// TIA Portal V20 program export: 1 tag tables, 4 data types, 5 data blocks, 8 code blocks (in call order from the OBs), 4 instance data blocks

VAR_GLOBAL   // PLC tag table "Default tag table"
   Tag_1 AT %I500.0 : Bool;
   Tag_2 AT %I500.1 : Bool;
   Tag_3 AT %I500.2 : Bool;
   Tag_4 AT %I500.3 : Bool;
   Tag_5 AT %I500.6 : Bool;
   Tag_6 AT %I500.7 : Bool;
   Tag_7 AT %I501.0 : Bool;
   Tag_8 AT %I501.1 : Bool;
   Tag_9 AT %I501.2 : Bool;
   Tag_10 AT %I501.3 : Bool;
   Tag_11 AT %I501.4 : Bool;
   Tag_12 AT %I501.5 : Bool;
   Tag_13 AT %I501.6 : Bool;
   Tag_14 AT %I501.7 : Bool;
   Tag_15 AT %I502.1 : Bool;
   Tag_16 AT %I502.2 : Bool;
   Tag_17 AT %I502.3 : Bool;
   Tag_18 AT %I502.4 : Bool;
   Tag_19 AT %I502.5 : Bool;
   Tag_20 AT %I502.6 : Bool;
   Tag_21 AT %I502.7 : Bool;
   Tag_22 AT %I503.0 : Bool;
   Tag_23 AT %I503.1 : Bool;
   Tag_24 AT %I503.2 : Bool;
   Tag_25 AT %I503.3 : Bool;
   Tag_26 AT %I503.4 : Bool;
   Tag_41 AT %IW508 : Word;
   Tag_42 AT %IW528 : Word;
   Tag_43 AT %IW532 : Word;
   Tag_44 AT %IW650 : Word;
   Tag_45 AT %IW64 : Word;
   Tag_46 AT %IW66 : Word;
   Tag_47 AT %IW68 : Word;
   Tag_48 AT %IW70 : Word;
   Tag_49 AT %IW72 : Word;
   Tag_50 AT %IW74 : Word;
   Tag_51 AT %IW76 : Word;
   Tag_52 AT %IW78 : Word;
   Tag_27 AT %Q500.0 : Bool;
   Tag_28 AT %Q500.1 : Bool;
   Tag_29 AT %Q500.2 : Bool;
   Tag_30 AT %Q500.4 : Bool;
   Tag_31 AT %Q500.5 : Bool;
   Tag_32 AT %Q501.0 : Bool;
   Tag_33 AT %Q501.1 : Bool;
   Tag_34 AT %Q501.2 : Bool;
   Tag_35 AT %Q501.3 : Bool;
   Tag_36 AT %Q501.4 : Bool;
   Tag_37 AT %Q501.5 : Bool;
   Tag_38 AT %Q502.0 : Bool;
   Tag_39 AT %Q502.1 : Bool;
   Tag_40 AT %Q502.2 : Bool;
   Tag_53 AT %QW64 : Word;
   Tag_54 AT %QW66 : Word;
   "Clock_0.5Hz" AT %M0.7 : Bool;
   AirStarWord0IN AT %IW80 : Word;
   AirStarWord2IN AT %IW82 : Word;
   AirStarWord0OUT AT %QW68 : Word;
   AirStarWord2OUT AT %QW70 : Word;
   FirstScan AT %M1.0 : Bool;
   AlwaysTrue AT %M1.2 : Bool;
   DI1_SYS_ControlHealthy AT %I0.0 : Bool;   // Safety/control circuit healthy
   DI2_SPR_1 AT %I0.1 : Bool;   // Spare (wired to -X3:1)
   DI3_SYS_CycleStart AT %I0.2 : Bool;   // Cycle start pushbutton (local/remote)
   DI4_SYS_CycleStop AT %I0.3 : Bool;   // Cycle stop pushbutton (NC)
   DI5_SHR_RunFwdFB AT %I0.4 : Bool;   // Shredder running forward feedback
   DI6_SHR_RunRevFB AT %I0.5 : Bool;   // Shredder running reverse feedback
   DI7_SYS_MotorFault AT %I0.6 : Bool;   // Motor fault (soft start fault relay)
   DI8_HPR_LevelHigh AT %I0.7 : Bool;   // Hopper high level sensor
   DI9_IFC_Running AT %I1.0 : Bool;   // Infeed conveyor running feedback
   DI10_DIS_Running AT %I1.1 : Bool;   // Discharge conveyor running feedback
   DI11_PSH_PowerPackRunning AT %I1.2 : Bool;   // Pusher power pack running feedback
   DI12_PSH_HomeLimit AT %I1.3 : Bool;   // Pusher parked/home position
   DI13_PSH_FullTravelLimit AT %I1.4 : Bool;   // Pusher fully extended position
   DI14_PSH_HighPressure AT %I1.5 : Bool;   // Pusher hydraulic high pressure switch
   DI15_SYS_DownstreamRunning AT %I2.0 : Bool;   // Downstream equipment running
   DI16_PSH_LocalRemote AT %I2.1 : Bool;   // Pusher operation local/remote selector
   DI17_SPR_2 AT %I2.2 : Bool;   // Spare (wired to terminal)
   DI18_SPR_3 AT %I2.3 : Bool;   // Spare (wired to terminal)
   DI19_SPR_4 AT %I2.4 : Bool;   // Spare (wired to terminal)
   DI20_SPR_5 AT %I2.5 : Bool;   // Spare (wired to terminal)
   DI21_SPR_6 AT %I2.6 : Bool;   // Spare (wired to terminal)
   DI22_SPR_7 AT %I2.7 : Bool;   // Spare (wired to terminal)
   DQ1_SHR_RunFwd AT %Q0.0 : Bool;   // Run shredder forward command
   DQ2_SHR_RunRev AT %Q0.1 : Bool;   // Run shredder reverse command
   DQ3_PSH_RunPowerPack AT %Q0.2 : Bool;   // Run pusher power pack command
   DQ4_IFC_Run AT %Q0.3 : Bool;   // Run infeed conveyor command
   DQ5_DIS_Run AT %Q0.4 : Bool;   // Run discharge conveyor command
   DQ6_PSH_Extend AT %Q0.5 : Bool;   // Pusher extend solenoid command
   DQ7_PSH_Retract AT %Q0.6 : Bool;   // Pusher retract solenoid command
   DQ8_SYS_InCycle AT %Q0.7 : Bool;   // Machine in-cycle status
   DQ9_SYS_EnableUpstream AT %Q1.0 : Bool;   // Enable upstream equipment (volt-free)
   DQ10_SYS_PreStartSounder AT %Q1.1 : Bool;   // Pre-start warning sounder/beacon
   DQ11_SHR_FaultReset AT %Q2.0 : Bool;   // Soft start motor fault reset
   DQ12_SPR_1 AT %Q2.1 : Bool;   // Spare (relay fitted)
   DQ13_SPR_2 AT %Q2.2 : Bool;   // Spare (relay fitted)
   DQ14_SPR_3 AT %Q2.3 : Bool;   // Spare (relay fitted)
   DQ15_SPR_4 AT %Q2.4 : Bool;   // Spare (relay fitted)
   DQ16_SPR_5 AT %Q2.5 : Bool;   // Spare (relay fitted)
   DQ17_SPR_6 AT %Q2.6 : Bool;   // Spare (wired to -X13:6)
   DQ18_SPR_7 AT %Q2.7 : Bool;   // Spare (wired to -X13:7)
END_VAR

TYPE "MotorFwdRevIOSet"
// stored: IsFailsafeCompliant false
   STRUCT
      InHand : Bool;
      AutoStartSignal : Bool;
      HandStartSignal : Bool;
      RunningFBFwd : Bool;
      RunningFBRev : Bool;
      FaultFB : Bool;
      SystemHealthy : Bool;
      PreStartDone : Bool;
      InhibitMotor : Bool;
      FaultReset : Bool;
      FTTime : Real;
      EnableUPSTime : Real;
      FaultActive : Bool;
      RunFwd : Bool;
      RunRev : Bool;
      UPSEnable : Bool;
      FTR : Bool;
      FTS : Bool;
      HrsRun : UDInt;
      Telemetry : Int;
      Alarm : Word;
      "Name" : String;
      HandIntervention : Bool;
      RecentStart : Bool;
      TryRunMotor : Bool;
      Shutdown : Bool;
      ShutdownComplete : Bool;
      ShutdownTime : Real;
      StopMotor : Bool;
      ReverseDelay : Real;
      ReverseIgnoreFT : Real;
      Reverse : Bool;
      HandReverse : Bool;
   END_STRUCT;
END_TYPE

TYPE "UDT_HopperBlockageIO"
// Caller-visible interface (C-115) for FB_HopperBlockageMonitor. FC_ControlMain writes HopperLevelHigh/PlantRunning/FaultReset in and reads HopperBlockedAlarm/HopperBlockStopReq out (wiring is a separate integration step). Per the Gate-1 supervisory-monitor exemption (NEW-HBA-07) this pure monitor carries no enable/ready/running vocabulary stubs. BlockedTimeThreshold/ClearDebounceTime are this instance's own tunables (C-307), commissioning defaults set as the iDB start values.
// stored: IsFailsafeCompliant false
   STRUCT
      HopperLevelHigh : Bool;   // In (FC_ControlMain, from DB_Input.Hopper_Level_High at integration): hopper high-level sensor - the blockage condition this FB supervises for persistence.
      PlantRunning : Bool;   // In (FC_ControlMain, from DB_Input.Shredder_Run_Fwd_FB OR Shredder_Run_Rev_FB): plant-running gate - the persistence window accrues only while the plant actually runs (Q-HBA-04), so a full hopper at standstill never alarms.
      FaultReset : Bool;   // In (FC_ControlMain, from DB_Controls.FaultReset): shared operator reset - clears the latched alarm below. C-115 handshake vocabulary, verbatim across the corpus.
      BlockedTimeThreshold : Time;   // Setting: cumulative high-and-running persistence threshold, seconds (start value T#60S). FB-own tunable per C-307 (not a shared DB_Settings member), commissioning-set as the iDB start value.
      ClearDebounceTime : Time;   // Setting: confirmed-clear filter time, seconds (start value T#2S) - the hopper must read clear continuously this long before the window re-arms, rejecting sensor chatter (Q-HBA-02). FB-own tunable per C-307, commissioning-set.
      HopperBlockedAlarm : Bool;   // Out: latched hopper-blockage alarm (REQ-HBA-001/004). RETAIN - deliberately survives a power cycle (C-124 carve-out), cleared only by FaultReset, like the sequencer's DischargeConveyorTimeoutFault; a blockage needing a human still needs acknowledgement after a restart.
      HopperBlockStopReq : Bool;   // Out: stop/inhibit demand (Q-HBA-05) - tracks the latched alarm and, being RETAIN, correspondingly persists across a power cycle until acknowledged. The FB writes no shared tag; integration wires this demand to the actual stop separately.
   END_STRUCT;
END_TYPE

TYPE "UDT_PusherIO"
// stored: IsFailsafeCompliant false
   STRUCT
      "Step" : Int;
      Fitted : Bool;
      Enable : Bool;
      AutoStartSignal : Bool;   // In: C-115 handshake vocabulary (owner ruling 2026-07-17, task 09, resolution 2) - external run permission, caller-asserted, named after the site's real chained-permissive pattern (FB_MotorFwdRevSystem.IO.AutoStartSignal), not doc 06's illustrative name. Unwired by FC_ControlMain for now - no established caller need for this integration; C-115 requires the member regardless. Distinct from Enable above (FB-computed, Fitted AND Mode<>0) - that's this block's own internal readiness gate, not the external permission this member carries.
      Mode : Int;
      HopperHighLevel : Bool;
      ManualCycleCmd : Bool;
      ParkCmd : Bool;   // In (FC_ControlMain, from the sequencer's PusherParkCmd): plant pre-start park request - while set, an idle off-home ram reparks to home after the pre-motion warning (REQ-045). With a live cycle request, one of the only two repark occasions (owner ruling 2026-07-16); jog release deliberately leaves the ram where it stopped (REQ-039).
      CycleInhibit : Bool;   // In (FC_ControlMain, from the sequencer's PusherCycleInhibitCmd): the plant has a live stop reason - no cycle may launch (CycleRequest gated) and an in-flight cycle aborts to Retract and parks (CycleAbort). Hand-jog is deliberately exempt (owner amendment 2026-07-16, REQ-040): only the mode-0 force (stop button/unhealthy) blocks jogging.
      JogExtendCmd : Bool;
      JogRetractCmd : Bool;
      HomeLimit : Bool;
      FullTravelLimit : Bool;
      HighPressure : Bool;
      PowerPackRunningFB : Bool;
      FaultReset : Bool;
      EndTravelTimeout : Real;
      ParkedTimeout : Real;
      EndTravelHoldTime : Real;
      PumpRunOnTime : Real;
      JogWarningTime : Real;
      PressureTripConfirmTime : Real;
      PressureClearResumeDelay : Real;
      PressureTripCountThreshold : Int;
      Cycling : Bool;   // Out: this block's C-115 running-equivalent (owner ruling 2026-07-17, task 09 resolution 2) - Step <> 0. Already wired (NETWORK 13); recognized as satisfying C-115's running slot under this block's own established name rather than duplicated under the generic vocabulary.
      Blocked : Bool;
      EndTravelTimeoutFault : Bool;
      ParkedTimeoutFault : Bool;
      BothSwitchesFault : Bool;
      RunPowerPack : Bool;
      Extend : Bool;
      Retract : Bool;
      JogPreStartSounder : Bool;
   END_STRUCT;
END_TYPE

TYPE "UDT_ShredderSequencerIO"
// stored: IsFailsafeCompliant false
   STRUCT
      CycleStart : Bool;
      AutoStartSignal : Bool;   // In: C-115 handshake vocabulary (owner ruling 2026-07-17, task 09, resolution 2) - external run permission, caller-asserted, named after the site's real chained-permissive pattern (FB_MotorFwdRevSystem.IO.AutoStartSignal), not doc 06's illustrative name. Unwired by FC_ControlMain for now - CycleStart/CycleStop already carry this sequencer's actual start/stop triggering; C-115 requires the vocabulary member regardless of whether this integration uses it.
      CycleStop : Bool;
      DownstreamRunning : Bool;
      SystemHealthy : Bool;   // In (FC_ControlMain, from DB_Input.Control_Healthy): safety/control circuit healthy. Loss asserts StopCmd - every step aborts to Idle and a fresh CycleStart press is required after recovery, so an E-stop reset can never self-restart the plant (REQ-062).
      DischargeConvRunning : Bool;
      HopperLevelHigh : Bool;
      ShredderRunFwdFB : Bool;
      ShredderRunRevFB : Bool;   // In (FC_ControlMain, from DB_Input.Shredder_Run_Rev_FB): confirmed reverse-running feedback. Step 30's ReverseRunTimer times this, not bare step dwell, so ShredderReverseRunTime buys actual reverse rotation, not a motor-off pause (REQ-005).
      ShredderMotorCurrent : Real;
      MotorFaultActive : Bool;
      FaultReset : Bool;
      OperatorPusherMode : Int;
      PusherJogPreStartSounder : Bool;
      "Step" : Int;
      DischargeConveyorTimeoutFault : Bool;
      ShredderBlockedFault : Bool;
      RunDischargeConv : Bool;
      RunInfeedConv : Bool;
      EnableUpstream : Bool;   // Out: this sequencer's C-115 ready-equivalent (owner ruling 2026-07-17, task 09 resolution 2) - asserted once Step 50 (Running) has held long enough (UpstreamEnableTimer, NETWORK 11) that whatever's downstream may enable. Same role as FB_MotorFwdRevSystem.IO.UPSEnable under this project's own established name for this signal - not duplicated under the generic vocabulary name.
      PreStartSounder : Bool;
      InCycle : Bool;   // Out: this sequencer's C-115 running-equivalent (owner ruling 2026-07-17, task 09 resolution 2) - Step <> 0 (NETWORK 15), same shape as the pusher's own Cycling. Was previously an unwritten dead member (standing C-610 finding); wiring it to satisfy C-115's running slot closes that finding too.
      MotorReverseCmd : Bool;
      MotorAutoStartCmd : Bool;
      MotorPreStartDoneCmd : Bool;
      MotorStartArm : Bool;   // Out: asserted through PreStart (Step 10) only - one fresh, operator-commanded start attempt arms the motor once. FC_ControlMain ORs it into the imported motor FB's RecentStart, which that FB self-clears once running or faulted (its own press-to-arm contract), so no restart happens without a new cycle start (REQ-062).
      PusherModeCmd : Int;
      PusherParkCmd : Bool;   // Out: pre-start park request to the pusher - held through the machine-start steps 20-40 (range intent per C-603: any step inserted inside the start ramp still wants the pusher home) so the pusher reparks-with-warning if off home once the siren phase completes (REQ-045).
      PusherCycleInhibitCmd : Bool;   // Out: mirrors StopCmd - while the plant has any live stop reason (stop button, downstream lost, circuit unhealthy) the pusher must not launch or continue a cycle into the stopped plant (owner amendment 2026-07-16). Unlike the mode-0 force, this leaves hand-jog available: jog is blocked only by the stop button or an unhealthy circuit, never by downstream absence (REQ-040).
   END_STRUCT;
END_TYPE

DATA_BLOCK "DB_AnalogInput"   // DB9
{ S7_Optimized_Access := 'TRUE' }
VERSION : 0.1
// Analog local IO buffer - separate from DB_Input per C-304 (analog IO in its own dedicated DBs). No physical channel exists yet for ShredderMotorCurrent - no AI module in the hardware table this project was built from; stays unmapped (no FC_AnalogInputMap yet) until real hardware is confirmed, per the project owner's own 'genuine analog current feedback' decision.
// stored: AutoNumber true, DBAccessibleFromOPCUA true, IsOnlyStoredInLoadMemory false, IsRetainMemResEnabled false, IsWriteProtectedInAS false, MemoryReserve 100
   VAR
      ShredderMotorCurrent : Real;
   END_VAR
BEGIN
END_DATA_BLOCK

DATA_BLOCK "DB_Controls"   // DB4
{ S7_Optimized_Access := 'TRUE' }
VERSION : 0.1
// Operator/HMI command surface (C-306). Written by HMI, consumed by equipment FBs and the sequencer - not logic-internal state.
// stored: AutoNumber true, DBAccessibleFromOPCUA true, IsOnlyStoredInLoadMemory false, IsRetainMemResEnabled false, IsWriteProtectedInAS false, MemoryReserve 100
   VAR
      PusherMode : Int;
      PusherManualCycleCmd : Bool;
      PusherJogExtendCmd : Bool;
      PusherJogRetractCmd : Bool;
      FaultReset : Bool;
   END_VAR
BEGIN
END_DATA_BLOCK

DATA_BLOCK "DB_Input"   // DB1
{ S7_Optimized_Access := 'TRUE' }
VERSION : 0.1
// stored: AutoNumber true, DBAccessibleFromOPCUA true, IsOnlyStoredInLoadMemory false, IsRetainMemResEnabled false, IsWriteProtectedInAS false, MemoryReserve 100
   VAR
      Test : Array[0..22] of Bool;
      SpareDI : Array[1..7] of Bool;
      Control_Healthy : Bool;
      Cycle_Start : Bool;
      Cycle_Stop : Bool;
      Shredder_Run_Fwd_FB : Bool;
      Shredder_Run_Rev_FB : Bool;
      Motor_Fault : Bool;
      Hopper_Level_High : Bool;
      Infeed_Conv_Running : Bool;
      Discharge_Conv_Running : Bool;
      Pusher_PowerPack_Running : Bool;
      Pusher_Home_Limit : Bool;
      Pusher_Full_Travel_Limit : Bool;
      Pusher_High_Pressure : Bool;
      Downstream_Running : Bool;
      Pusher_Local_Remote : Bool;
   END_VAR
BEGIN
END_DATA_BLOCK

DATA_BLOCK "DB_PLC"   // DB7
{ S7_Optimized_Access := 'TRUE' }
VERSION : 0.1
// PLC-specific system data (C-305). Simulation is force-reset FALSE at every startup (OB100, C-305/C-403) regardless of retentivity - simulation mode must never survive a power cycle; start values only apply at download, not restart.
// stored: AutoNumber true, DBAccessibleFromOPCUA true, IsOnlyStoredInLoadMemory false, IsRetainMemResEnabled false, IsWriteProtectedInAS false, MemoryReserve 100
   VAR RETAIN
      Simulation : Bool := FALSE;
   END_VAR
BEGIN
END_DATA_BLOCK

DATA_BLOCK "DB_Settings"   // DB3
{ S7_Optimized_Access := 'TRUE' }
VERSION : 0.1
// Plant/system-level tunables (C-307) - HMI/operator writes, PLC read-only (C-308). Start values are commissioning defaults (C-309). Five formerly-unconfigured live-zero timings were given site-practice defaults and signed off 2026-07-16. The four overcurrent members remain deliberately unconfigured - see their own member comments.
// stored: AutoNumber true, DBAccessibleFromOPCUA true, IsOnlyStoredInLoadMemory false, IsRetainMemResEnabled false, IsWriteProtectedInAS false, MemoryReserve 100
   VAR RETAIN
      PreStartSounderTime : Real := 10.0;
      ShredderReverseRunTime : Real := 6.0;
      InfeedRestartDelay : Real := 5.0;
      InfeedToUpstreamEnableDelay : Real := 3.0;
      OvercurrentSetpointMedium : Real;   // Unconfigured by design: the overcurrent family is disarmed (no AI hardware, Q-11; per-machine-type values unresolved, Q-04). No number is proposed until the detection arms - setting one now would imply protection that does not exist.
      OvercurrentSetpointHigh : Real;   // Unconfigured by design - same basis as OvercurrentSetpointMedium (Q-11/Q-04).
      OvercurrentMediumDelay : Real;   // Unconfigured by design - same basis as OvercurrentSetpointMedium (Q-11/Q-04); no spec number exists either (Q-02).
      OvercurrentHighDelay : Real;   // Unconfigured by design - same basis as OvercurrentSetpointMedium (Q-11/Q-04); no spec number exists either (Q-02).
      OvercurrentSpinUpAllowance : Real := 3.0;
      ReversalRetryPauseTime : Real := 4.0;
      ReversalWindowTime : Real := 180.0;
      ReversalCountThreshold : Int := 5;
      PressureTripConfirmTime : Real := 0.5;
      PressureClearResumeDelay : Real := 5.0;
      PressureTripCountThreshold : Int := 5;
      PusherEndTravelTimeout : Real := 60.0;
      PusherParkedTimeout : Real := 30.0;
      PusherEndTravelHoldTime : Real := 2.0;
      PusherPumpRunOnTime : Real := 5.0;
      PusherJogWarningTime : Real := 1.0;
      PusherFitted : Bool := TRUE;
      DischargeConveyorTimeout : Real := 10.0;
   END_VAR
BEGIN
END_DATA_BLOCK

ORGANIZATION_BLOCK "Main"   // OB1, LAD, ProgramCycle
TITLE = "Main Program Sweep (Cycle)"
{ S7_Optimized_Access := 'TRUE' }
VERSION : 0.1
// stored: AutoNumber true, IsIECCheckEnabled false, SetENOAutomatically false
   VAR_INPUT
      Initial_Call : Bool;   // Initial call of this OB
      Remanence : Bool;   // =True, if remanent data are available
   END_VAR
BEGIN

REGION Network 1: Hopper-Blockage Stimulus Model
   // Advances the commanded timeline the hopper-blockage monitor is tested against and presents it to the input buffer's test members. It runs ahead of the input map because for a commanded input the model is the field: the map that follows chooses between the terminal and the test member, and it must find this scan's commanded state rather than the previous scan's. Outside a run it drives nothing and the map reads the field.
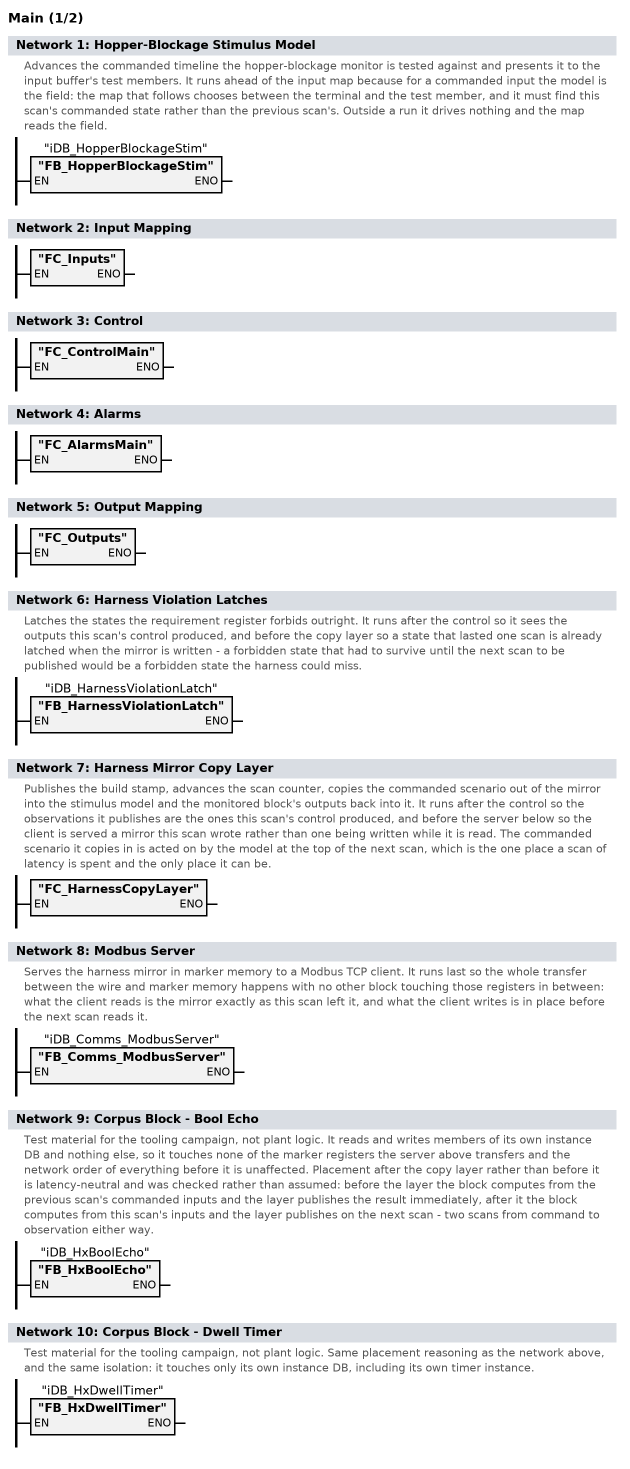
   RUNG wire#powerrail
      "iDB_HopperBlockageStim"()
   END_RUNG
   // the same network as SCL:
   "iDB_HopperBlockageStim"();   // "FB_HopperBlockageStim"
END_REGION

REGION Network 2: Input Mapping
   RUNG wire#powerrail
      "FC_Inputs"()
   END_RUNG
   // the same network as SCL:
   "FC_Inputs"();
END_REGION

REGION Network 3: Control
   RUNG wire#powerrail
      "FC_ControlMain"()
   END_RUNG
   // the same network as SCL:
   "FC_ControlMain"();
END_REGION

REGION Network 4: Alarms
   RUNG wire#powerrail
      "FC_AlarmsMain"()
   END_RUNG
   // the same network as SCL:
   "FC_AlarmsMain"();
END_REGION

REGION Network 5: Output Mapping
   RUNG wire#powerrail
      "FC_Outputs"()
   END_RUNG
   // the same network as SCL:
   "FC_Outputs"();
END_REGION

REGION Network 6: Harness Violation Latches
   // Latches the states the requirement register forbids outright. It runs after the control so it sees the outputs this scan's control produced, and before the copy layer so a state that lasted one scan is already latched when the mirror is written - a forbidden state that had to survive until the next scan to be published would be a forbidden state the harness could miss.
   RUNG wire#powerrail
      "iDB_HarnessViolationLatch"()
   END_RUNG
   // the same network as SCL:
   "iDB_HarnessViolationLatch"();   // "FB_HarnessViolationLatch"
END_REGION

REGION Network 7: Harness Mirror Copy Layer
   // Publishes the build stamp, advances the scan counter, copies the commanded scenario out of the mirror into the stimulus model and the monitored block's outputs back into it. It runs after the control so the observations it publishes are the ones this scan's control produced, and before the server below so the client is served a mirror this scan wrote rather than one being written while it is read. The commanded scenario it copies in is acted on by the model at the top of the next scan, which is the one place a scan of latency is spent and the only place it can be.
   RUNG wire#powerrail
      "FC_HarnessCopyLayer"()
   END_RUNG
   // the same network as SCL:
   "FC_HarnessCopyLayer"();
END_REGION

REGION Network 8: Modbus Server
   // Serves the harness mirror in marker memory to a Modbus TCP client. It runs last so the whole transfer between the wire and marker memory happens with no other block touching those registers in between: what the client reads is the mirror exactly as this scan left it, and what the client writes is in place before the next scan reads it.
   RUNG wire#powerrail
      "iDB_Comms_ModbusServer"()
   END_RUNG
   // the same network as SCL:
   "iDB_Comms_ModbusServer"();   // "FB_Comms_ModbusServer"
END_REGION

REGION Network 9: Corpus Block - Bool Echo
   // Test material for the tooling campaign, not plant logic. It reads and writes members of its own instance DB and nothing else, so it touches none of the marker registers the server above transfers and the network order of everything before it is unaffected. Placement after the copy layer rather than before it is latency-neutral and was checked rather than assumed: before the layer the block computes from the previous scan's commanded inputs and the layer publishes the result immediately, after it the block computes from this scan's inputs and the layer publishes on the next scan - two scans from command to observation either way.
   RUNG wire#powerrail
      "iDB_HxBoolEcho"()
   END_RUNG
   // the same network as SCL:
   "iDB_HxBoolEcho"();   // "FB_HxBoolEcho"
END_REGION

REGION Network 10: Corpus Block - Dwell Timer
   // Test material for the tooling campaign, not plant logic. Same placement reasoning as the network above, and the same isolation: it touches only its own instance DB, including its own timer instance.
   RUNG wire#powerrail
      "iDB_HxDwellTimer"()
   END_RUNG
   // the same network as SCL:
   "iDB_HxDwellTimer"();   // "FB_HxDwellTimer"
END_REGION

REGION Network 11: Corpus Block - Int Sum
   // Test material for the tooling campaign, not plant logic. Same placement reasoning as the networks above, and the same isolation: it touches only its own instance DB.
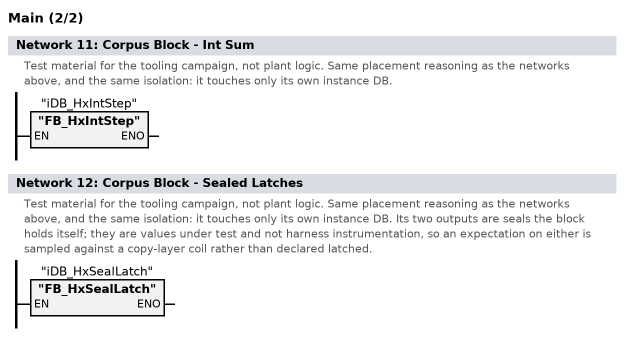
   RUNG wire#powerrail
      "iDB_HxIntStep"()
   END_RUNG
   // the same network as SCL:
   "iDB_HxIntStep"();   // "FB_HxIntStep"
END_REGION

REGION Network 12: Corpus Block - Sealed Latches
   // Test material for the tooling campaign, not plant logic. Same placement reasoning as the networks above, and the same isolation: it touches only its own instance DB. Its two outputs are seals the block holds itself; they are values under test and not harness instrumentation, so an expectation on either is sampled against a copy-layer coil rather than declared latched.
   RUNG wire#powerrail
      "iDB_HxSealLatch"()
   END_RUNG
   // the same network as SCL:
   "iDB_HxSealLatch"();   // "FB_HxSealLatch"
END_REGION
END_ORGANIZATION_BLOCK

FUNCTION "FC_Inputs" : Void   // FC1, LAD
TITLE = Input Map
{ S7_Optimized_Access := 'TRUE' }
VERSION : 0.1
// stored: AutoNumber true, IsIECCheckEnabled false, SetENOAutomatically false, UDAEnableTagReadback false
BEGIN

REGION Network 1: PLC1 Built-in DI (CPU 1214C)
   // DI4_SYS_CycleStop is a normally-closed pushbutton: negated at this map layer so DB_Input.Cycle_Stop reads active-high (true = operator commanding stop) like every other buffer member - the input-mapping pattern's negated variant. Field polarity is absorbed here only; logic never compensates (C-304).
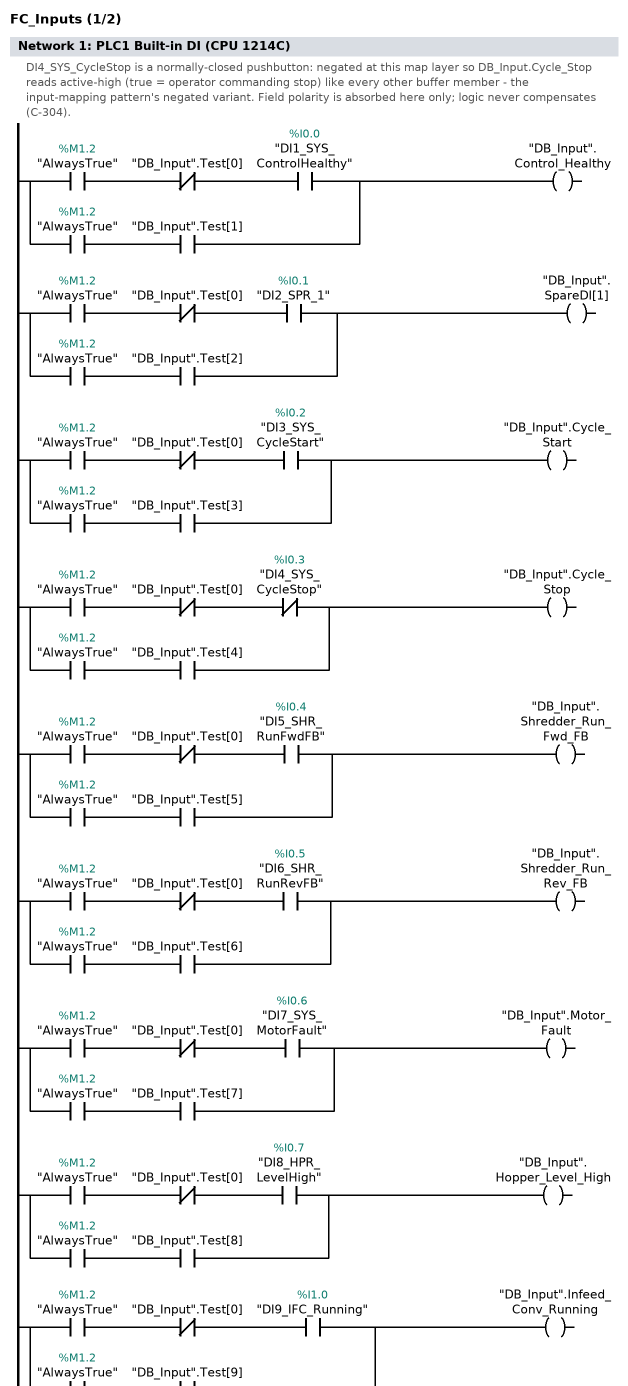
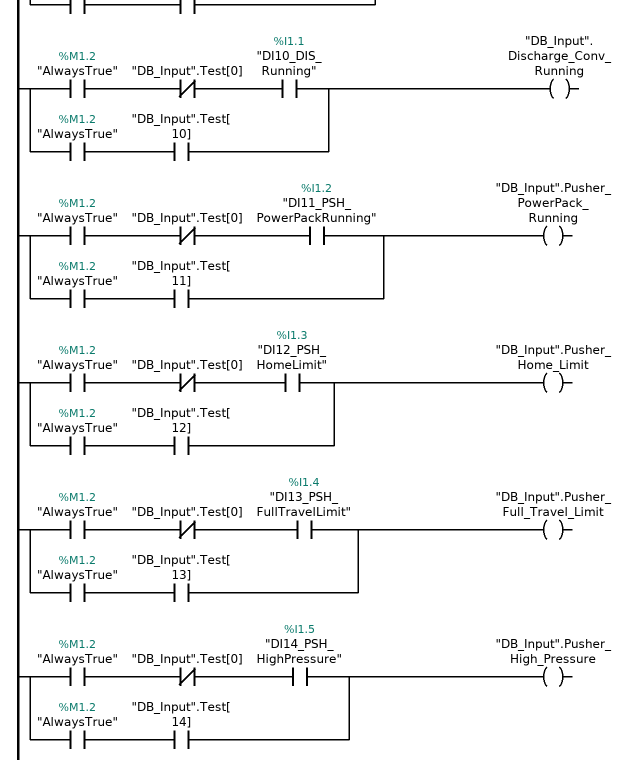
   RUNG wire#powerrail
      Contact( "AlwaysTrue" )
      I_Contact( "DB_Input".Test[0] )
      Contact( "DI1_SYS_ControlHealthy" )
      wire#w1
      Coil( "DB_Input".Control_Healthy )
   END_RUNG
   RUNG wire#powerrail
      Contact( "AlwaysTrue" )
      Contact( "DB_Input".Test[1] )
   END_RUNG wire#w1
   RUNG wire#powerrail
      Contact( "AlwaysTrue" )
      I_Contact( "DB_Input".Test[0] )
      Contact( "DI2_SPR_1" )
      wire#w2
      Coil( "DB_Input".SpareDI[1] )
   END_RUNG
   RUNG wire#powerrail
      Contact( "AlwaysTrue" )
      Contact( "DB_Input".Test[2] )
   END_RUNG wire#w2
   RUNG wire#powerrail
      Contact( "AlwaysTrue" )
      I_Contact( "DB_Input".Test[0] )
      Contact( "DI3_SYS_CycleStart" )
      wire#w3
      Coil( "DB_Input".Cycle_Start )
   END_RUNG
   RUNG wire#powerrail
      Contact( "AlwaysTrue" )
      Contact( "DB_Input".Test[3] )
   END_RUNG wire#w3
   RUNG wire#powerrail
      Contact( "AlwaysTrue" )
      I_Contact( "DB_Input".Test[0] )
      I_Contact( "DI4_SYS_CycleStop" )
      wire#w4
      Coil( "DB_Input".Cycle_Stop )
   END_RUNG
   RUNG wire#powerrail
      Contact( "AlwaysTrue" )
      Contact( "DB_Input".Test[4] )
   END_RUNG wire#w4
   RUNG wire#powerrail
      Contact( "AlwaysTrue" )
      I_Contact( "DB_Input".Test[0] )
      Contact( "DI5_SHR_RunFwdFB" )
      wire#w5
      Coil( "DB_Input".Shredder_Run_Fwd_FB )
   END_RUNG
   RUNG wire#powerrail
      Contact( "AlwaysTrue" )
      Contact( "DB_Input".Test[5] )
   END_RUNG wire#w5
   RUNG wire#powerrail
      Contact( "AlwaysTrue" )
      I_Contact( "DB_Input".Test[0] )
      Contact( "DI6_SHR_RunRevFB" )
      wire#w6
      Coil( "DB_Input".Shredder_Run_Rev_FB )
   END_RUNG
   RUNG wire#powerrail
      Contact( "AlwaysTrue" )
      Contact( "DB_Input".Test[6] )
   END_RUNG wire#w6
   RUNG wire#powerrail
      Contact( "AlwaysTrue" )
      I_Contact( "DB_Input".Test[0] )
      Contact( "DI7_SYS_MotorFault" )
      wire#w7
      Coil( "DB_Input".Motor_Fault )
   END_RUNG
   RUNG wire#powerrail
      Contact( "AlwaysTrue" )
      Contact( "DB_Input".Test[7] )
   END_RUNG wire#w7
   RUNG wire#powerrail
      Contact( "AlwaysTrue" )
      I_Contact( "DB_Input".Test[0] )
      Contact( "DI8_HPR_LevelHigh" )
      wire#w8
      Coil( "DB_Input".Hopper_Level_High )
   END_RUNG
   RUNG wire#powerrail
      Contact( "AlwaysTrue" )
      Contact( "DB_Input".Test[8] )
   END_RUNG wire#w8
   RUNG wire#powerrail
      Contact( "AlwaysTrue" )
      I_Contact( "DB_Input".Test[0] )
      Contact( "DI9_IFC_Running" )
      wire#w9
      Coil( "DB_Input".Infeed_Conv_Running )
   END_RUNG
   RUNG wire#powerrail
      Contact( "AlwaysTrue" )
      Contact( "DB_Input".Test[9] )
   END_RUNG wire#w9
   RUNG wire#powerrail
      Contact( "AlwaysTrue" )
      I_Contact( "DB_Input".Test[0] )
      Contact( "DI10_DIS_Running" )
      wire#w10
      Coil( "DB_Input".Discharge_Conv_Running )
   END_RUNG
   RUNG wire#powerrail
      Contact( "AlwaysTrue" )
      Contact( "DB_Input".Test[10] )
   END_RUNG wire#w10
   RUNG wire#powerrail
      Contact( "AlwaysTrue" )
      I_Contact( "DB_Input".Test[0] )
      Contact( "DI11_PSH_PowerPackRunning" )
      wire#w11
      Coil( "DB_Input".Pusher_PowerPack_Running )
   END_RUNG
   RUNG wire#powerrail
      Contact( "AlwaysTrue" )
      Contact( "DB_Input".Test[11] )
   END_RUNG wire#w11
   RUNG wire#powerrail
      Contact( "AlwaysTrue" )
      I_Contact( "DB_Input".Test[0] )
      Contact( "DI12_PSH_HomeLimit" )
      wire#w12
      Coil( "DB_Input".Pusher_Home_Limit )
   END_RUNG
   RUNG wire#powerrail
      Contact( "AlwaysTrue" )
      Contact( "DB_Input".Test[12] )
   END_RUNG wire#w12
   RUNG wire#powerrail
      Contact( "AlwaysTrue" )
      I_Contact( "DB_Input".Test[0] )
      Contact( "DI13_PSH_FullTravelLimit" )
      wire#w13
      Coil( "DB_Input".Pusher_Full_Travel_Limit )
   END_RUNG
   RUNG wire#powerrail
      Contact( "AlwaysTrue" )
      Contact( "DB_Input".Test[13] )
   END_RUNG wire#w13
   RUNG wire#powerrail
      Contact( "AlwaysTrue" )
      I_Contact( "DB_Input".Test[0] )
      Contact( "DI14_PSH_HighPressure" )
      wire#w14
      Coil( "DB_Input".Pusher_High_Pressure )
   END_RUNG
   RUNG wire#powerrail
      Contact( "AlwaysTrue" )
      Contact( "DB_Input".Test[14] )
   END_RUNG wire#w14
   // the same network as SCL:
   "DB_Input".Control_Healthy := ("AlwaysTrue" AND NOT "DB_Input".Test[0] AND "DI1_SYS_ControlHealthy") OR ("AlwaysTrue" AND "DB_Input".Test[1]);
   "DB_Input".SpareDI[1] := ("AlwaysTrue" AND NOT "DB_Input".Test[0] AND "DI2_SPR_1") OR ("AlwaysTrue" AND "DB_Input".Test[2]);
   "DB_Input".Cycle_Start := ("AlwaysTrue" AND NOT "DB_Input".Test[0] AND "DI3_SYS_CycleStart") OR ("AlwaysTrue" AND "DB_Input".Test[3]);
   "DB_Input".Cycle_Stop := ("AlwaysTrue" AND NOT "DB_Input".Test[0] AND NOT "DI4_SYS_CycleStop") OR ("AlwaysTrue" AND "DB_Input".Test[4]);
   "DB_Input".Shredder_Run_Fwd_FB := ("AlwaysTrue" AND NOT "DB_Input".Test[0] AND "DI5_SHR_RunFwdFB") OR ("AlwaysTrue" AND "DB_Input".Test[5]);
   "DB_Input".Shredder_Run_Rev_FB := ("AlwaysTrue" AND NOT "DB_Input".Test[0] AND "DI6_SHR_RunRevFB") OR ("AlwaysTrue" AND "DB_Input".Test[6]);
   "DB_Input".Motor_Fault := ("AlwaysTrue" AND NOT "DB_Input".Test[0] AND "DI7_SYS_MotorFault") OR ("AlwaysTrue" AND "DB_Input".Test[7]);
   "DB_Input".Hopper_Level_High := ("AlwaysTrue" AND NOT "DB_Input".Test[0] AND "DI8_HPR_LevelHigh") OR ("AlwaysTrue" AND "DB_Input".Test[8]);
   "DB_Input".Infeed_Conv_Running := ("AlwaysTrue" AND NOT "DB_Input".Test[0] AND "DI9_IFC_Running") OR ("AlwaysTrue" AND "DB_Input".Test[9]);
   "DB_Input".Discharge_Conv_Running := ("AlwaysTrue" AND NOT "DB_Input".Test[0] AND "DI10_DIS_Running") OR ("AlwaysTrue" AND "DB_Input".Test[10]);
   "DB_Input".Pusher_PowerPack_Running := ("AlwaysTrue" AND NOT "DB_Input".Test[0] AND "DI11_PSH_PowerPackRunning") OR ("AlwaysTrue" AND "DB_Input".Test[11]);
   "DB_Input".Pusher_Home_Limit := ("AlwaysTrue" AND NOT "DB_Input".Test[0] AND "DI12_PSH_HomeLimit") OR ("AlwaysTrue" AND "DB_Input".Test[12]);
   "DB_Input".Pusher_Full_Travel_Limit := ("AlwaysTrue" AND NOT "DB_Input".Test[0] AND "DI13_PSH_FullTravelLimit") OR ("AlwaysTrue" AND "DB_Input".Test[13]);
   "DB_Input".Pusher_High_Pressure := ("AlwaysTrue" AND NOT "DB_Input".Test[0] AND "DI14_PSH_HighPressure") OR ("AlwaysTrue" AND "DB_Input".Test[14]);
END_REGION

REGION Network 2: PLC1.1 SM1223 DI
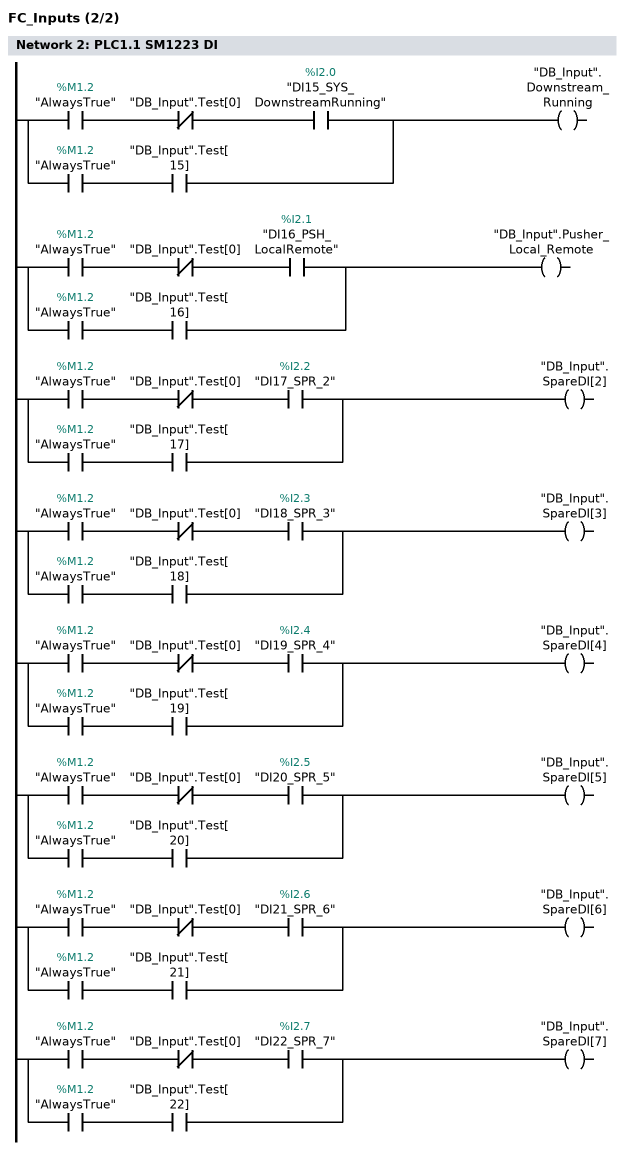
   RUNG wire#powerrail
      Contact( "AlwaysTrue" )
      I_Contact( "DB_Input".Test[0] )
      Contact( "DI15_SYS_DownstreamRunning" )
      wire#w1
      Coil( "DB_Input".Downstream_Running )
   END_RUNG
   RUNG wire#powerrail
      Contact( "AlwaysTrue" )
      Contact( "DB_Input".Test[15] )
   END_RUNG wire#w1
   RUNG wire#powerrail
      Contact( "AlwaysTrue" )
      I_Contact( "DB_Input".Test[0] )
      Contact( "DI16_PSH_LocalRemote" )
      wire#w2
      Coil( "DB_Input".Pusher_Local_Remote )
   END_RUNG
   RUNG wire#powerrail
      Contact( "AlwaysTrue" )
      Contact( "DB_Input".Test[16] )
   END_RUNG wire#w2
   RUNG wire#powerrail
      Contact( "AlwaysTrue" )
      I_Contact( "DB_Input".Test[0] )
      Contact( "DI17_SPR_2" )
      wire#w3
      Coil( "DB_Input".SpareDI[2] )
   END_RUNG
   RUNG wire#powerrail
      Contact( "AlwaysTrue" )
      Contact( "DB_Input".Test[17] )
   END_RUNG wire#w3
   RUNG wire#powerrail
      Contact( "AlwaysTrue" )
      I_Contact( "DB_Input".Test[0] )
      Contact( "DI18_SPR_3" )
      wire#w4
      Coil( "DB_Input".SpareDI[3] )
   END_RUNG
   RUNG wire#powerrail
      Contact( "AlwaysTrue" )
      Contact( "DB_Input".Test[18] )
   END_RUNG wire#w4
   RUNG wire#powerrail
      Contact( "AlwaysTrue" )
      I_Contact( "DB_Input".Test[0] )
      Contact( "DI19_SPR_4" )
      wire#w5
      Coil( "DB_Input".SpareDI[4] )
   END_RUNG
   RUNG wire#powerrail
      Contact( "AlwaysTrue" )
      Contact( "DB_Input".Test[19] )
   END_RUNG wire#w5
   RUNG wire#powerrail
      Contact( "AlwaysTrue" )
      I_Contact( "DB_Input".Test[0] )
      Contact( "DI20_SPR_5" )
      wire#w6
      Coil( "DB_Input".SpareDI[5] )
   END_RUNG
   RUNG wire#powerrail
      Contact( "AlwaysTrue" )
      Contact( "DB_Input".Test[20] )
   END_RUNG wire#w6
   RUNG wire#powerrail
      Contact( "AlwaysTrue" )
      I_Contact( "DB_Input".Test[0] )
      Contact( "DI21_SPR_6" )
      wire#w7
      Coil( "DB_Input".SpareDI[6] )
   END_RUNG
   RUNG wire#powerrail
      Contact( "AlwaysTrue" )
      Contact( "DB_Input".Test[21] )
   END_RUNG wire#w7
   RUNG wire#powerrail
      Contact( "AlwaysTrue" )
      I_Contact( "DB_Input".Test[0] )
      Contact( "DI22_SPR_7" )
      wire#w8
      Coil( "DB_Input".SpareDI[7] )
   END_RUNG
   RUNG wire#powerrail
      Contact( "AlwaysTrue" )
      Contact( "DB_Input".Test[22] )
   END_RUNG wire#w8
   // the same network as SCL:
   "DB_Input".Downstream_Running := ("AlwaysTrue" AND NOT "DB_Input".Test[0] AND "DI15_SYS_DownstreamRunning") OR ("AlwaysTrue" AND "DB_Input".Test[15]);
   "DB_Input".Pusher_Local_Remote := ("AlwaysTrue" AND NOT "DB_Input".Test[0] AND "DI16_PSH_LocalRemote") OR ("AlwaysTrue" AND "DB_Input".Test[16]);
   "DB_Input".SpareDI[2] := ("AlwaysTrue" AND NOT "DB_Input".Test[0] AND "DI17_SPR_2") OR ("AlwaysTrue" AND "DB_Input".Test[17]);
   "DB_Input".SpareDI[3] := ("AlwaysTrue" AND NOT "DB_Input".Test[0] AND "DI18_SPR_3") OR ("AlwaysTrue" AND "DB_Input".Test[18]);
   "DB_Input".SpareDI[4] := ("AlwaysTrue" AND NOT "DB_Input".Test[0] AND "DI19_SPR_4") OR ("AlwaysTrue" AND "DB_Input".Test[19]);
   "DB_Input".SpareDI[5] := ("AlwaysTrue" AND NOT "DB_Input".Test[0] AND "DI20_SPR_5") OR ("AlwaysTrue" AND "DB_Input".Test[20]);
   "DB_Input".SpareDI[6] := ("AlwaysTrue" AND NOT "DB_Input".Test[0] AND "DI21_SPR_6") OR ("AlwaysTrue" AND "DB_Input".Test[21]);
   "DB_Input".SpareDI[7] := ("AlwaysTrue" AND NOT "DB_Input".Test[0] AND "DI22_SPR_7") OR ("AlwaysTrue" AND "DB_Input".Test[22]);
END_REGION
END_FUNCTION

FUNCTION "FC_ControlMain" : Void   // FC3, LAD
TITLE = Control Main
{ S7_Optimized_Access := 'TRUE' }
VERSION : 0.1
// Control area-Main (C-109): every cross-instance fact in the project lives here (C-127) - buffer-to-instance input wiring, the sequencer/motor/pusher calls in dependency order (sequencer decides, motor and pusher obey within the same scan), inter-instance command wiring, and the buffer output map. No working logic beyond wiring, with two documented extras (C-606): the In_Cycle lamp OR (owner ruling 2026-07-16, REQ-069 - field feedbacks, not commands) and the soft-start fault-reset pass-through to DQ11 (panel provides the output; Q-14 records the open control-on question).
// stored: AutoNumber true, IsIECCheckEnabled false, SetENOAutomatically false, UDAEnableTagReadback false
BEGIN

REGION Network 1: Sequencer Input Wiring
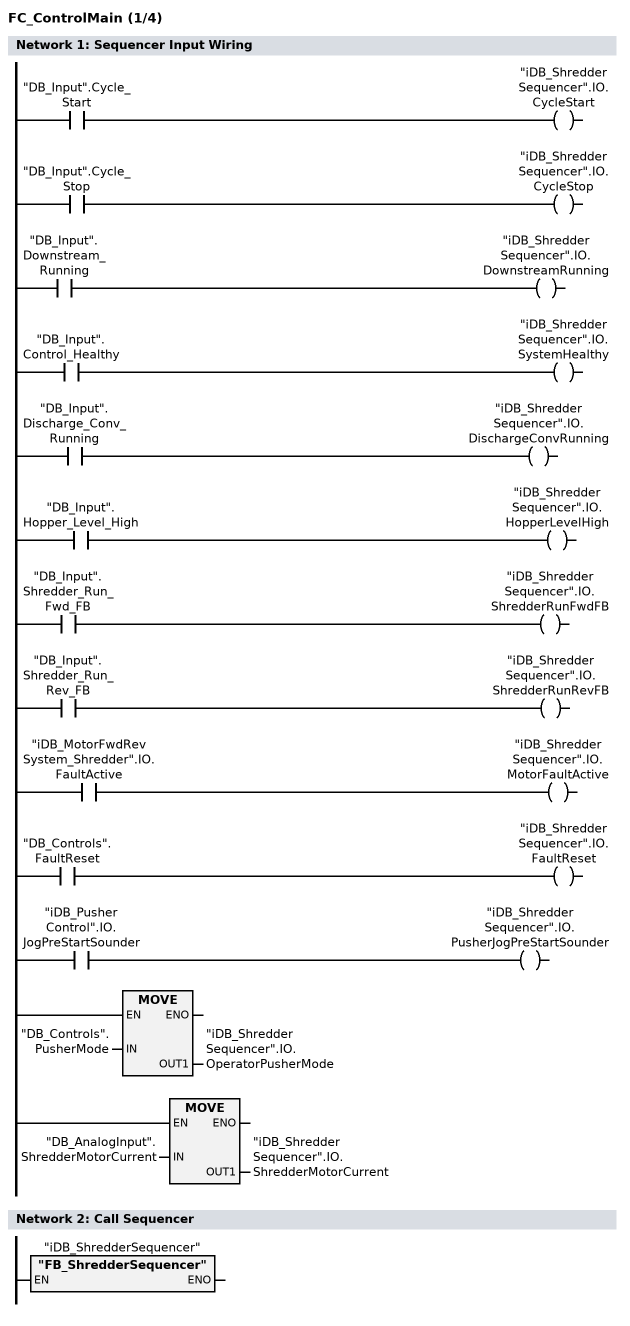
   RUNG wire#powerrail
      Contact( "DB_Input".Cycle_Start )
      Coil( "iDB_ShredderSequencer".IO.CycleStart )
   END_RUNG
   RUNG wire#powerrail
      Contact( "DB_Input".Cycle_Stop )
      Coil( "iDB_ShredderSequencer".IO.CycleStop )
   END_RUNG
   RUNG wire#powerrail
      Contact( "DB_Input".Downstream_Running )
      Coil( "iDB_ShredderSequencer".IO.DownstreamRunning )
   END_RUNG
   RUNG wire#powerrail
      Contact( "DB_Input".Control_Healthy )
      Coil( "iDB_ShredderSequencer".IO.SystemHealthy )
   END_RUNG
   RUNG wire#powerrail
      Contact( "DB_Input".Discharge_Conv_Running )
      Coil( "iDB_ShredderSequencer".IO.DischargeConvRunning )
   END_RUNG
   RUNG wire#powerrail
      Contact( "DB_Input".Hopper_Level_High )
      Coil( "iDB_ShredderSequencer".IO.HopperLevelHigh )
   END_RUNG
   RUNG wire#powerrail
      Contact( "DB_Input".Shredder_Run_Fwd_FB )
      Coil( "iDB_ShredderSequencer".IO.ShredderRunFwdFB )
   END_RUNG
   RUNG wire#powerrail
      Contact( "DB_Input".Shredder_Run_Rev_FB )
      Coil( "iDB_ShredderSequencer".IO.ShredderRunRevFB )
   END_RUNG
   RUNG wire#powerrail
      Contact( "iDB_MotorFwdRevSystem_Shredder".IO.FaultActive )
      Coil( "iDB_ShredderSequencer".IO.MotorFaultActive )
   END_RUNG
   RUNG wire#powerrail
      Contact( "DB_Controls".FaultReset )
      Coil( "iDB_ShredderSequencer".IO.FaultReset )
   END_RUNG
   RUNG wire#powerrail
      Contact( "iDB_PusherControl".IO.JogPreStartSounder )
      Coil( "iDB_ShredderSequencer".IO.PusherJogPreStartSounder )
   END_RUNG
   RUNG wire#powerrail
      Move(in := "DB_Controls".PusherMode, out1 => "iDB_ShredderSequencer".IO.OperatorPusherMode)
   END_RUNG
   RUNG wire#powerrail
      Move(in := "DB_AnalogInput".ShredderMotorCurrent, out1 => "iDB_ShredderSequencer".IO.ShredderMotorCurrent)
   END_RUNG
   // the same network as SCL:
   "iDB_ShredderSequencer".IO.CycleStart := "DB_Input".Cycle_Start;
   "iDB_ShredderSequencer".IO.CycleStop := "DB_Input".Cycle_Stop;
   "iDB_ShredderSequencer".IO.DownstreamRunning := "DB_Input".Downstream_Running;
   "iDB_ShredderSequencer".IO.SystemHealthy := "DB_Input".Control_Healthy;
   "iDB_ShredderSequencer".IO.DischargeConvRunning := "DB_Input".Discharge_Conv_Running;
   "iDB_ShredderSequencer".IO.HopperLevelHigh := "DB_Input".Hopper_Level_High;
   "iDB_ShredderSequencer".IO.ShredderRunFwdFB := "DB_Input".Shredder_Run_Fwd_FB;
   "iDB_ShredderSequencer".IO.ShredderRunRevFB := "DB_Input".Shredder_Run_Rev_FB;
   "iDB_ShredderSequencer".IO.MotorFaultActive := "iDB_MotorFwdRevSystem_Shredder".IO.FaultActive;
   "iDB_ShredderSequencer".IO.FaultReset := "DB_Controls".FaultReset;
   "iDB_ShredderSequencer".IO.PusherJogPreStartSounder := "iDB_PusherControl".IO.JogPreStartSounder;
   "iDB_ShredderSequencer".IO.OperatorPusherMode := "DB_Controls".PusherMode;
   "iDB_ShredderSequencer".IO.ShredderMotorCurrent := "DB_AnalogInput".ShredderMotorCurrent;
END_REGION

REGION Network 2: Call Sequencer
   RUNG wire#powerrail
      "iDB_ShredderSequencer"()
   END_RUNG
   // the same network as SCL:
   "iDB_ShredderSequencer"();   // "FB_ShredderSequencer"
END_REGION

REGION Network 3: MotorFwdRevSystem Wiring
   // InHand, InhibitMotor, and HandReverse are deliberate constants (C-604): unrequested imported-FB capability (hand mode, external inhibit, hand-reverse) carried disabled - design, not placeholder debt. RecentStart is armed, never driven: the sequencer's MotorStartArm (PreStart step only) ORs into the FB's own bit, and the FB's self-clear (once running or faulted - its N4 'set on start press' contract) is the only clearer, so one fresh start press arms exactly one start attempt and an E-stop or fault can never auto-restart the motor (REQ-062; replaces the RecentStart := AlwaysTrue strap that defeated the FB's semantics).
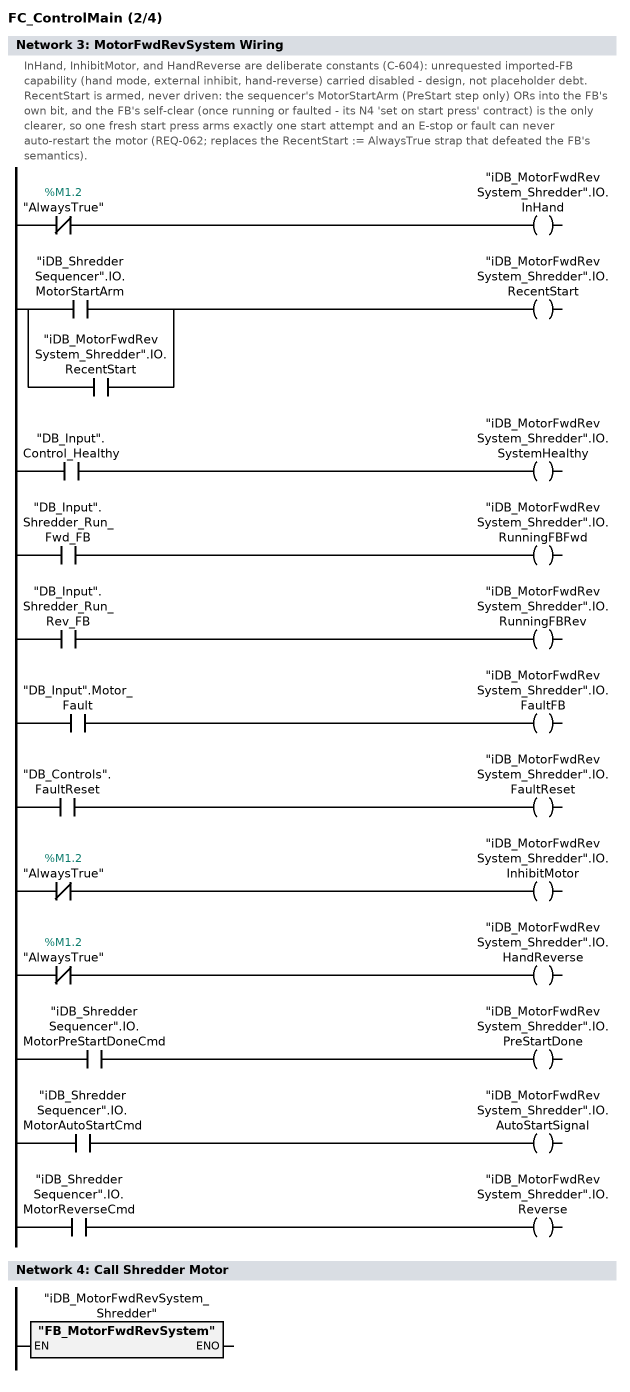
   RUNG wire#powerrail
      I_Contact( "AlwaysTrue" )
      Coil( "iDB_MotorFwdRevSystem_Shredder".IO.InHand )
   END_RUNG
   RUNG wire#powerrail
      Contact( "iDB_ShredderSequencer".IO.MotorStartArm )
      wire#w1
      Coil( "iDB_MotorFwdRevSystem_Shredder".IO.RecentStart )
   END_RUNG
   RUNG wire#powerrail
      Contact( "iDB_MotorFwdRevSystem_Shredder".IO.RecentStart )
   END_RUNG wire#w1
   RUNG wire#powerrail
      Contact( "DB_Input".Control_Healthy )
      Coil( "iDB_MotorFwdRevSystem_Shredder".IO.SystemHealthy )
   END_RUNG
   RUNG wire#powerrail
      Contact( "DB_Input".Shredder_Run_Fwd_FB )
      Coil( "iDB_MotorFwdRevSystem_Shredder".IO.RunningFBFwd )
   END_RUNG
   RUNG wire#powerrail
      Contact( "DB_Input".Shredder_Run_Rev_FB )
      Coil( "iDB_MotorFwdRevSystem_Shredder".IO.RunningFBRev )
   END_RUNG
   RUNG wire#powerrail
      Contact( "DB_Input".Motor_Fault )
      Coil( "iDB_MotorFwdRevSystem_Shredder".IO.FaultFB )
   END_RUNG
   RUNG wire#powerrail
      Contact( "DB_Controls".FaultReset )
      Coil( "iDB_MotorFwdRevSystem_Shredder".IO.FaultReset )
   END_RUNG
   RUNG wire#powerrail
      I_Contact( "AlwaysTrue" )
      Coil( "iDB_MotorFwdRevSystem_Shredder".IO.InhibitMotor )
   END_RUNG
   RUNG wire#powerrail
      I_Contact( "AlwaysTrue" )
      Coil( "iDB_MotorFwdRevSystem_Shredder".IO.HandReverse )
   END_RUNG
   RUNG wire#powerrail
      Contact( "iDB_ShredderSequencer".IO.MotorPreStartDoneCmd )
      Coil( "iDB_MotorFwdRevSystem_Shredder".IO.PreStartDone )
   END_RUNG
   RUNG wire#powerrail
      Contact( "iDB_ShredderSequencer".IO.MotorAutoStartCmd )
      Coil( "iDB_MotorFwdRevSystem_Shredder".IO.AutoStartSignal )
   END_RUNG
   RUNG wire#powerrail
      Contact( "iDB_ShredderSequencer".IO.MotorReverseCmd )
      Coil( "iDB_MotorFwdRevSystem_Shredder".IO.Reverse )
   END_RUNG
   // the same network as SCL:
   "iDB_MotorFwdRevSystem_Shredder".IO.InHand := NOT "AlwaysTrue";
   "iDB_MotorFwdRevSystem_Shredder".IO.RecentStart := "iDB_ShredderSequencer".IO.MotorStartArm OR "iDB_MotorFwdRevSystem_Shredder".IO.RecentStart;
   "iDB_MotorFwdRevSystem_Shredder".IO.SystemHealthy := "DB_Input".Control_Healthy;
   "iDB_MotorFwdRevSystem_Shredder".IO.RunningFBFwd := "DB_Input".Shredder_Run_Fwd_FB;
   "iDB_MotorFwdRevSystem_Shredder".IO.RunningFBRev := "DB_Input".Shredder_Run_Rev_FB;
   "iDB_MotorFwdRevSystem_Shredder".IO.FaultFB := "DB_Input".Motor_Fault;
   "iDB_MotorFwdRevSystem_Shredder".IO.FaultReset := "DB_Controls".FaultReset;
   "iDB_MotorFwdRevSystem_Shredder".IO.InhibitMotor := NOT "AlwaysTrue";
   "iDB_MotorFwdRevSystem_Shredder".IO.HandReverse := NOT "AlwaysTrue";
   "iDB_MotorFwdRevSystem_Shredder".IO.PreStartDone := "iDB_ShredderSequencer".IO.MotorPreStartDoneCmd;
   "iDB_MotorFwdRevSystem_Shredder".IO.AutoStartSignal := "iDB_ShredderSequencer".IO.MotorAutoStartCmd;
   "iDB_MotorFwdRevSystem_Shredder".IO.Reverse := "iDB_ShredderSequencer".IO.MotorReverseCmd;
END_REGION

REGION Network 4: Call Shredder Motor
   RUNG wire#powerrail
      "iDB_MotorFwdRevSystem_Shredder"()
   END_RUNG
   // the same network as SCL:
   "iDB_MotorFwdRevSystem_Shredder"();   // "FB_MotorFwdRevSystem"
END_REGION

REGION Network 5: PusherControl Wiring
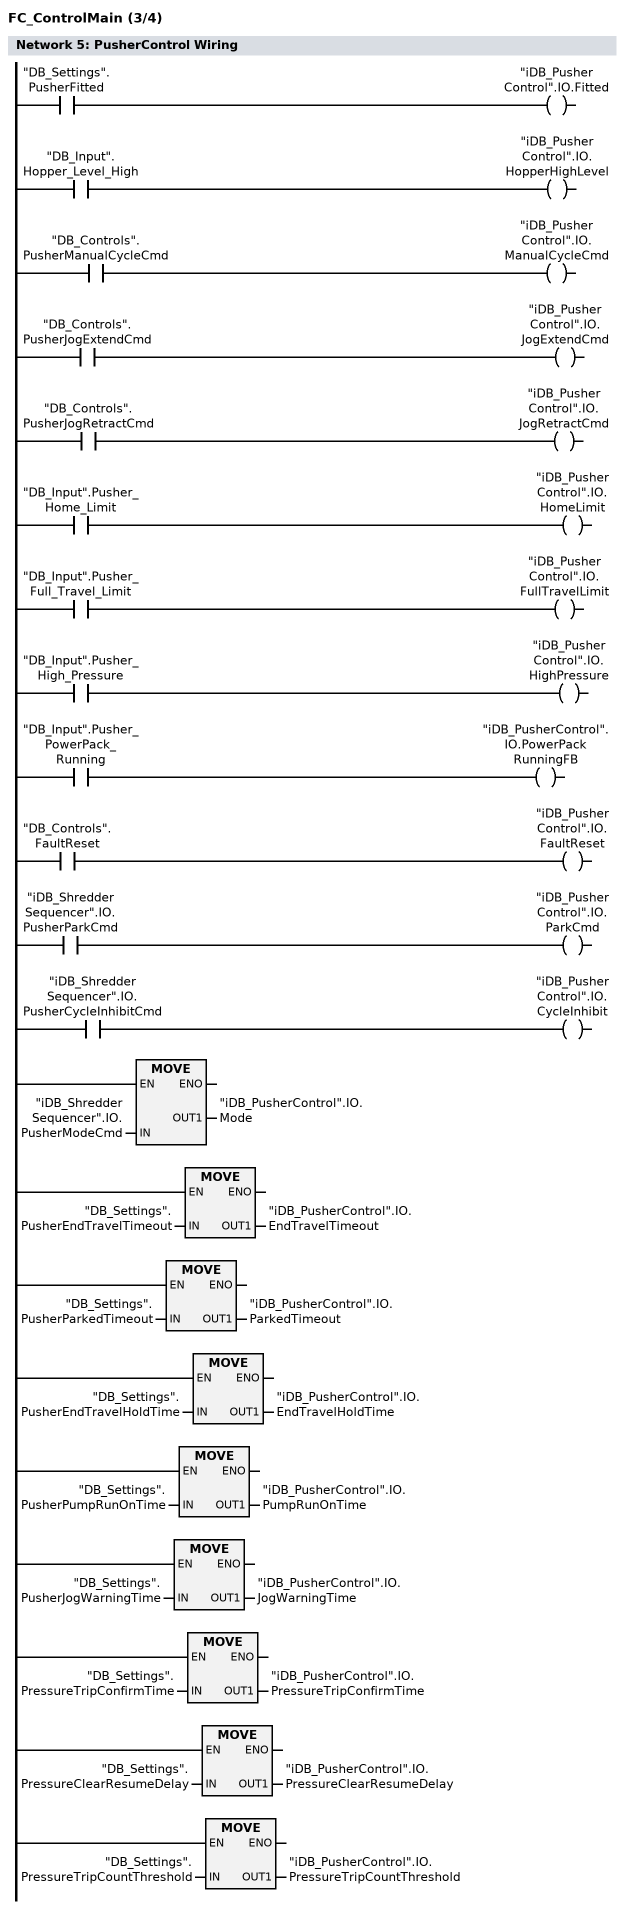
   RUNG wire#powerrail
      Contact( "DB_Settings".PusherFitted )
      Coil( "iDB_PusherControl".IO.Fitted )
   END_RUNG
   RUNG wire#powerrail
      Contact( "DB_Input".Hopper_Level_High )
      Coil( "iDB_PusherControl".IO.HopperHighLevel )
   END_RUNG
   RUNG wire#powerrail
      Contact( "DB_Controls".PusherManualCycleCmd )
      Coil( "iDB_PusherControl".IO.ManualCycleCmd )
   END_RUNG
   RUNG wire#powerrail
      Contact( "DB_Controls".PusherJogExtendCmd )
      Coil( "iDB_PusherControl".IO.JogExtendCmd )
   END_RUNG
   RUNG wire#powerrail
      Contact( "DB_Controls".PusherJogRetractCmd )
      Coil( "iDB_PusherControl".IO.JogRetractCmd )
   END_RUNG
   RUNG wire#powerrail
      Contact( "DB_Input".Pusher_Home_Limit )
      Coil( "iDB_PusherControl".IO.HomeLimit )
   END_RUNG
   RUNG wire#powerrail
      Contact( "DB_Input".Pusher_Full_Travel_Limit )
      Coil( "iDB_PusherControl".IO.FullTravelLimit )
   END_RUNG
   RUNG wire#powerrail
      Contact( "DB_Input".Pusher_High_Pressure )
      Coil( "iDB_PusherControl".IO.HighPressure )
   END_RUNG
   RUNG wire#powerrail
      Contact( "DB_Input".Pusher_PowerPack_Running )
      Coil( "iDB_PusherControl".IO.PowerPackRunningFB )
   END_RUNG
   RUNG wire#powerrail
      Contact( "DB_Controls".FaultReset )
      Coil( "iDB_PusherControl".IO.FaultReset )
   END_RUNG
   RUNG wire#powerrail
      Contact( "iDB_ShredderSequencer".IO.PusherParkCmd )
      Coil( "iDB_PusherControl".IO.ParkCmd )
   END_RUNG
   RUNG wire#powerrail
      Contact( "iDB_ShredderSequencer".IO.PusherCycleInhibitCmd )
      Coil( "iDB_PusherControl".IO.CycleInhibit )
   END_RUNG
   RUNG wire#powerrail
      Move(in := "iDB_ShredderSequencer".IO.PusherModeCmd, out1 => "iDB_PusherControl".IO.Mode)
   END_RUNG
   RUNG wire#powerrail
      Move(in := "DB_Settings".PusherEndTravelTimeout, out1 => "iDB_PusherControl".IO.EndTravelTimeout)
   END_RUNG
   RUNG wire#powerrail
      Move(in := "DB_Settings".PusherParkedTimeout, out1 => "iDB_PusherControl".IO.ParkedTimeout)
   END_RUNG
   RUNG wire#powerrail
      Move(in := "DB_Settings".PusherEndTravelHoldTime, out1 => "iDB_PusherControl".IO.EndTravelHoldTime)
   END_RUNG
   RUNG wire#powerrail
      Move(in := "DB_Settings".PusherPumpRunOnTime, out1 => "iDB_PusherControl".IO.PumpRunOnTime)
   END_RUNG
   RUNG wire#powerrail
      Move(in := "DB_Settings".PusherJogWarningTime, out1 => "iDB_PusherControl".IO.JogWarningTime)
   END_RUNG
   RUNG wire#powerrail
      Move(in := "DB_Settings".PressureTripConfirmTime, out1 => "iDB_PusherControl".IO.PressureTripConfirmTime)
   END_RUNG
   RUNG wire#powerrail
      Move(in := "DB_Settings".PressureClearResumeDelay, out1 => "iDB_PusherControl".IO.PressureClearResumeDelay)
   END_RUNG
   RUNG wire#powerrail
      Move(in := "DB_Settings".PressureTripCountThreshold, out1 => "iDB_PusherControl".IO.PressureTripCountThreshold)
   END_RUNG
   // the same network as SCL:
   "iDB_PusherControl".IO.Fitted := "DB_Settings".PusherFitted;
   "iDB_PusherControl".IO.HopperHighLevel := "DB_Input".Hopper_Level_High;
   "iDB_PusherControl".IO.ManualCycleCmd := "DB_Controls".PusherManualCycleCmd;
   "iDB_PusherControl".IO.JogExtendCmd := "DB_Controls".PusherJogExtendCmd;
   "iDB_PusherControl".IO.JogRetractCmd := "DB_Controls".PusherJogRetractCmd;
   "iDB_PusherControl".IO.HomeLimit := "DB_Input".Pusher_Home_Limit;
   "iDB_PusherControl".IO.FullTravelLimit := "DB_Input".Pusher_Full_Travel_Limit;
   "iDB_PusherControl".IO.HighPressure := "DB_Input".Pusher_High_Pressure;
   "iDB_PusherControl".IO.PowerPackRunningFB := "DB_Input".Pusher_PowerPack_Running;
   "iDB_PusherControl".IO.FaultReset := "DB_Controls".FaultReset;
   "iDB_PusherControl".IO.ParkCmd := "iDB_ShredderSequencer".IO.PusherParkCmd;
   "iDB_PusherControl".IO.CycleInhibit := "iDB_ShredderSequencer".IO.PusherCycleInhibitCmd;
   "iDB_PusherControl".IO.Mode := "iDB_ShredderSequencer".IO.PusherModeCmd;
   "iDB_PusherControl".IO.EndTravelTimeout := "DB_Settings".PusherEndTravelTimeout;
   "iDB_PusherControl".IO.ParkedTimeout := "DB_Settings".PusherParkedTimeout;
   "iDB_PusherControl".IO.EndTravelHoldTime := "DB_Settings".PusherEndTravelHoldTime;
   "iDB_PusherControl".IO.PumpRunOnTime := "DB_Settings".PusherPumpRunOnTime;
   "iDB_PusherControl".IO.JogWarningTime := "DB_Settings".PusherJogWarningTime;
   "iDB_PusherControl".IO.PressureTripConfirmTime := "DB_Settings".PressureTripConfirmTime;
   "iDB_PusherControl".IO.PressureClearResumeDelay := "DB_Settings".PressureClearResumeDelay;
   "iDB_PusherControl".IO.PressureTripCountThreshold := "DB_Settings".PressureTripCountThreshold;
END_REGION

REGION Network 6: Call Pusher
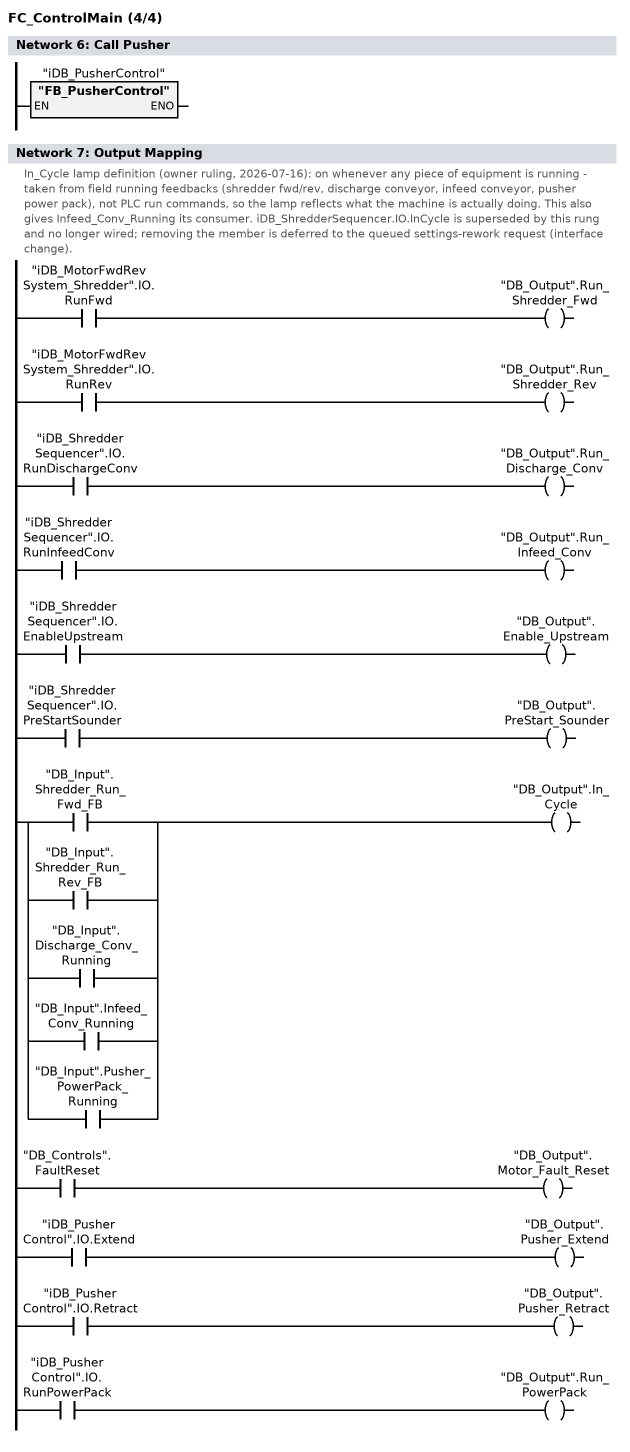
   RUNG wire#powerrail
      "iDB_PusherControl"()
   END_RUNG
   // the same network as SCL:
   "iDB_PusherControl"();   // "FB_PusherControl"
END_REGION

REGION Network 7: Output Mapping
   // In_Cycle lamp definition (owner ruling, 2026-07-16): on whenever any piece of equipment is running - taken from field running feedbacks (shredder fwd/rev, discharge conveyor, infeed conveyor, pusher power pack), not PLC run commands, so the lamp reflects what the machine is actually doing. This also gives Infeed_Conv_Running its consumer. iDB_ShredderSequencer.IO.InCycle is superseded by this rung and no longer wired; removing the member is deferred to the queued settings-rework request (interface change).
   RUNG wire#powerrail
      Contact( "iDB_MotorFwdRevSystem_Shredder".IO.RunFwd )
      Coil( "DB_Output".Run_Shredder_Fwd )
   END_RUNG
   RUNG wire#powerrail
      Contact( "iDB_MotorFwdRevSystem_Shredder".IO.RunRev )
      Coil( "DB_Output".Run_Shredder_Rev )
   END_RUNG
   RUNG wire#powerrail
      Contact( "iDB_ShredderSequencer".IO.RunDischargeConv )
      Coil( "DB_Output".Run_Discharge_Conv )
   END_RUNG
   RUNG wire#powerrail
      Contact( "iDB_ShredderSequencer".IO.RunInfeedConv )
      Coil( "DB_Output".Run_Infeed_Conv )
   END_RUNG
   RUNG wire#powerrail
      Contact( "iDB_ShredderSequencer".IO.EnableUpstream )
      Coil( "DB_Output".Enable_Upstream )
   END_RUNG
   RUNG wire#powerrail
      Contact( "iDB_ShredderSequencer".IO.PreStartSounder )
      Coil( "DB_Output".PreStart_Sounder )
   END_RUNG
   RUNG wire#powerrail
      Contact( "DB_Input".Shredder_Run_Fwd_FB )
      wire#w1
      Coil( "DB_Output".In_Cycle )
   END_RUNG
   RUNG wire#powerrail
      Contact( "DB_Input".Shredder_Run_Rev_FB )
   END_RUNG wire#w1
   RUNG wire#powerrail
      Contact( "DB_Input".Discharge_Conv_Running )
   END_RUNG wire#w1
   RUNG wire#powerrail
      Contact( "DB_Input".Infeed_Conv_Running )
   END_RUNG wire#w1
   RUNG wire#powerrail
      Contact( "DB_Input".Pusher_PowerPack_Running )
   END_RUNG wire#w1
   RUNG wire#powerrail
      Contact( "DB_Controls".FaultReset )
      Coil( "DB_Output".Motor_Fault_Reset )
   END_RUNG
   RUNG wire#powerrail
      Contact( "iDB_PusherControl".IO.Extend )
      Coil( "DB_Output".Pusher_Extend )
   END_RUNG
   RUNG wire#powerrail
      Contact( "iDB_PusherControl".IO.Retract )
      Coil( "DB_Output".Pusher_Retract )
   END_RUNG
   RUNG wire#powerrail
      Contact( "iDB_PusherControl".IO.RunPowerPack )
      Coil( "DB_Output".Run_PowerPack )
   END_RUNG
   // the same network as SCL:
   "DB_Output".Run_Shredder_Fwd := "iDB_MotorFwdRevSystem_Shredder".IO.RunFwd;
   "DB_Output".Run_Shredder_Rev := "iDB_MotorFwdRevSystem_Shredder".IO.RunRev;
   "DB_Output".Run_Discharge_Conv := "iDB_ShredderSequencer".IO.RunDischargeConv;
   "DB_Output".Run_Infeed_Conv := "iDB_ShredderSequencer".IO.RunInfeedConv;
   "DB_Output".Enable_Upstream := "iDB_ShredderSequencer".IO.EnableUpstream;
   "DB_Output".PreStart_Sounder := "iDB_ShredderSequencer".IO.PreStartSounder;
   "DB_Output".In_Cycle := "DB_Input".Shredder_Run_Fwd_FB OR "DB_Input".Shredder_Run_Rev_FB OR "DB_Input".Discharge_Conv_Running OR "DB_Input".Infeed_Conv_Running OR "DB_Input".Pusher_PowerPack_Running;
   "DB_Output".Motor_Fault_Reset := "DB_Controls".FaultReset;
   "DB_Output".Pusher_Extend := "iDB_PusherControl".IO.Extend;
   "DB_Output".Pusher_Retract := "iDB_PusherControl".IO.Retract;
   "DB_Output".Run_PowerPack := "iDB_PusherControl".IO.RunPowerPack;
END_REGION
END_FUNCTION

FUNCTION_BLOCK "FB_ShredderSequencer"   // FB8, LAD
TITLE = Shredder Plant Sequencer
{ S7_Optimized_Access := 'TRUE' }
VERSION : 0.1
// Shredder plant sequencer: commands the shredder motor (via FB_MotorFwdRevSystem, wired at FC_ControlMain) and gates infeed/discharge conveyors and upstream enable, through a stepped cycle. Step legend: 0=Idle (stopped, waiting for a start condition) - 10=PreStart (siren warning before motion; arms the motor via MotorStartArm) - 20=DischargeStart (discharge conveyor starting, timed) - 30=ReverseRun (reverse commanded; the motor FB's own ReverseDelay entry pause elapses inside this step, then ReverseRunTimer counts ShredderReverseRunTime of CONFIRMED reverse feedback) - 40=WaitForwardRun (waiting for forward-run feedback) - 50=Running (normal production; infeed/upstream-enable timers and overcurrent detection are live) - 60=OvercurrentAbort (tripped - pause, then retry into ReverseRun, or stay out if too many reversals). Stop-all (REQ-012/013/062): StopCmd = stop button OR downstream lost OR control circuit unhealthy - aborts every step to Idle. Pusher handling is split: stop button/unhealthy force pusher mode 0 (parks AND blocks jog), while any live stop reason - downstream loss included - raises PusherCycleInhibitCmd (no cycle launches or continues into a stopped plant, hand-jog stays available).
// stored: AutoNumber true, IsIECCheckEnabled false, IsRetainMemResEnabled false, MemoryReserve 100, SetENOAutomatically false, UDAEnableTagReadback false
   VAR RETAIN
      IO { S7_SetPoint := 'True'} : "UDT_ShredderSequencerIO";   // Caller-visible interface - every signal into or out of this block crosses here, nothing bypasses it: FC_ControlMain writes CycleStart/CycleStop/feedback/tunables in, reads Run*/EnableUpstream/PreStartSounder/motor-command bits out. See the block header for the Step value legend.
   END_VAR
   VAR
      StopCmd : Bool;   // Stop-all: operator CycleStop, loss of DownstreamRunning (nowhere for shredded material to go), or loss of SystemHealthy (control circuit/E-stop - REQ-062: recovery must demand a fresh start press, so the sequence may not sit in a run step through an E-stop). Read by every step's own stop transition below and mirrored to the pusher as PusherCycleInhibitCmd.
      PusherModeForceOff : Bool;   // The hard pusher force - operator stop or circuit-unhealthy, plus the overcurrent-abort step. Forces PusherModeCmd to 0, which parks the pusher AND blocks jogging. Deliberately narrower than the full StopCmd: downstream absence must leave hand-jog available (REQ-040), so it reaches the pusher only as PusherCycleInhibitCmd.
      ReversalWindowTimeMS : DInt;
      PreStartSounderTimeMS : DInt;
      DischargeConveyorTimeoutMS : DInt;
      ShredderReverseRunTimeMS : DInt;
      InfeedRestartDelayMS : DInt;
      InfeedToUpstreamEnableDelayMS : DInt;
      OvercurrentSpinUpAllowanceMS : DInt;
      OvercurrentMediumDelayMS : DInt;
      OvercurrentHighDelayMS : DInt;
      ReversalRetryPauseTimeMS : DInt;
      ReversalWindowTimer { S7_SetPoint := 'True'} : TON_TIME;
      ReversalStepEdge : Bool;
      ReversalStepEdgeMem : Bool;
      ReversalCount : Int;   // Reversals since the window last re-armed (not per-cycle, unlike the pusher's own PressureTripCount) - ReversalWindowTimer restarts the window every time this is above zero, so ReversalCountThreshold reversals must occur within one ReversalWindowTime of each other to raise ShredderBlockedFault, not just ReversalCountThreshold times ever.
      PreStartTimer { S7_SetPoint := 'True'} : TON_TIME;
      DischargeStartTimer { S7_SetPoint := 'True'} : TON_TIME;
      ReverseRunTimer { S7_SetPoint := 'True'} : TON_TIME;
      InfeedRestartTimer { S7_SetPoint := 'True'} : TON_TIME;
      UpstreamEnableTimer { S7_SetPoint := 'True'} : TON_TIME;
      InfeedRunning : Bool;   // Latched once InfeedRestartTimer has timed out from the last hopper-clear - drives RunInfeedConv directly and (after a further UpstreamEnableTimer delay) EnableUpstream.
      SpinUpTimer { S7_SetPoint := 'True'} : TON_TIME;
      OvercurrentMediumTimer { S7_SetPoint := 'True'} : TON_TIME;
      OvercurrentHighTimer { S7_SetPoint := 'True'} : TON_TIME;
      OvercurrentTripped : Bool;   // KNOWN GAP, not wired to real current yet: both timers below are gated 'AND NOT AlwaysTrue' (permanently false placeholders) because DB_AnalogInput.ShredderMotorCurrent > DB_Settings.OvercurrentSetpointMedium/High is a genuine Real-vs-Real comparison this converter's synthesizer can't type correctly yet (hardcodes Int). This bit, and Step 50's own overcurrent-abort transition, are dead code until that's built.
      OvercurrentAbortPauseTimer { S7_SetPoint := 'True'} : TON_TIME;
   END_VAR
   VAR_TEMP
      "Time" : Real;
   END_VAR
BEGIN

REGION Network 1: Stop Command
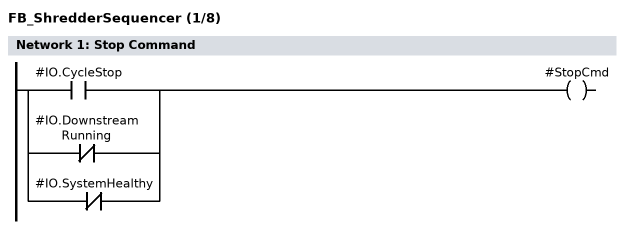
   RUNG wire#powerrail
      Contact( #IO.CycleStop )
      wire#w1
      Coil( #StopCmd )
   END_RUNG
   RUNG wire#powerrail
      I_Contact( #IO.DownstreamRunning )
   END_RUNG wire#w1
   RUNG wire#powerrail
      I_Contact( #IO.SystemHealthy )
   END_RUNG wire#w1
   // the same network as SCL:
   #StopCmd := #IO.CycleStop OR NOT #IO.DownstreamRunning OR NOT #IO.SystemHealthy;
END_REGION

REGION Network 2: HMI Time Conversions
   // HMI/DB_Settings times are Real seconds for operator legibility; every TON below needs its PT in DInt ms - one MUL+CONVERT pair per timer, matching the MotorDOL FTTime/EnableUPSTime idiom. All ten pairs sit together up front, so the x1000 conversion is done once per timer and reads the same way for every one of them.
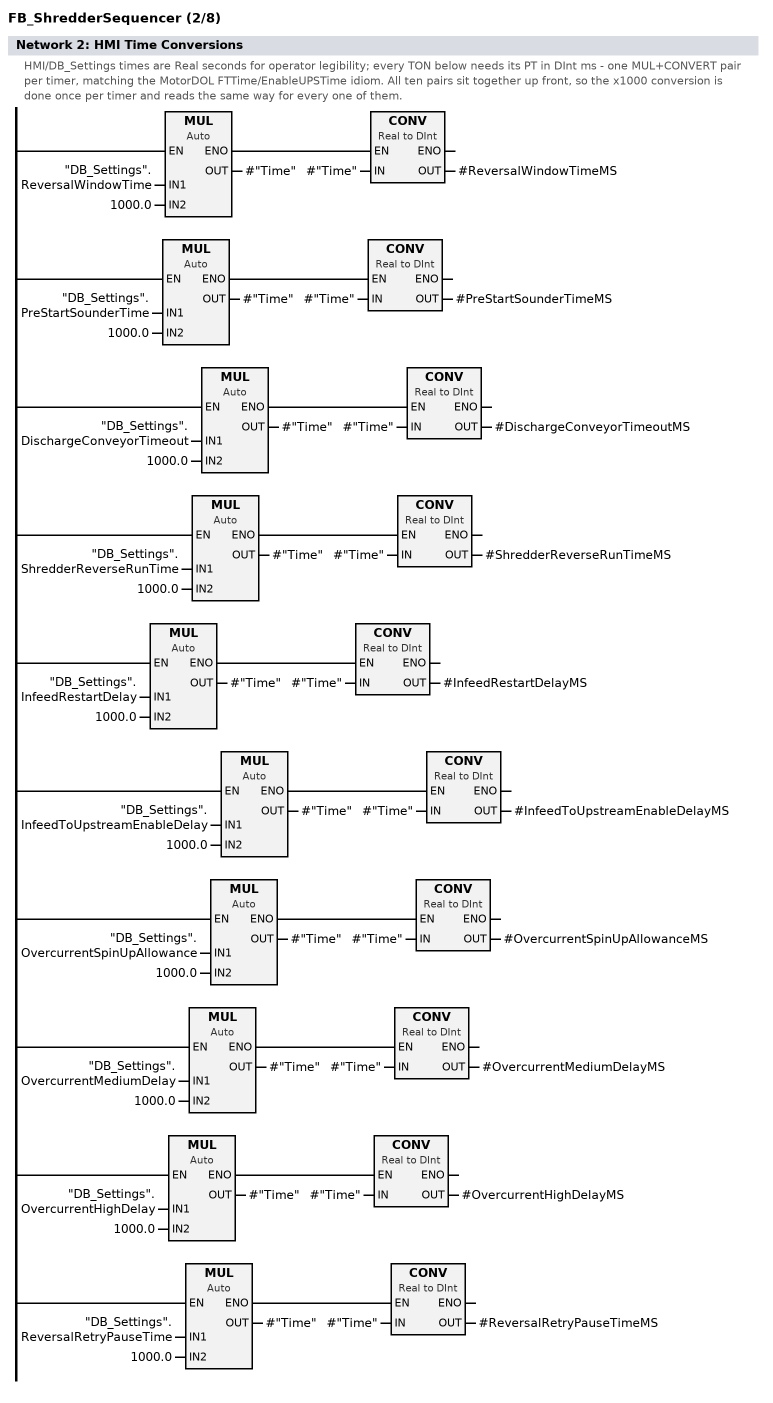
   RUNG wire#powerrail
      Mul(in1 := "DB_Settings".ReversalWindowTime, in2 := 1000.0, out => #"Time")
      { S7_Templates := "[SrcType := Real, DestType := DInt]" } Convert(in := #"Time", out => #ReversalWindowTimeMS)
   END_RUNG
   RUNG wire#powerrail
      Mul(in1 := "DB_Settings".PreStartSounderTime, in2 := 1000.0, out => #"Time")
      { S7_Templates := "[SrcType := Real, DestType := DInt]" } Convert(in := #"Time", out => #PreStartSounderTimeMS)
   END_RUNG
   RUNG wire#powerrail
      Mul(in1 := "DB_Settings".DischargeConveyorTimeout, in2 := 1000.0, out => #"Time")
      { S7_Templates := "[SrcType := Real, DestType := DInt]" } Convert(in := #"Time", out => #DischargeConveyorTimeoutMS)
   END_RUNG
   RUNG wire#powerrail
      Mul(in1 := "DB_Settings".ShredderReverseRunTime, in2 := 1000.0, out => #"Time")
      { S7_Templates := "[SrcType := Real, DestType := DInt]" } Convert(in := #"Time", out => #ShredderReverseRunTimeMS)
   END_RUNG
   RUNG wire#powerrail
      Mul(in1 := "DB_Settings".InfeedRestartDelay, in2 := 1000.0, out => #"Time")
      { S7_Templates := "[SrcType := Real, DestType := DInt]" } Convert(in := #"Time", out => #InfeedRestartDelayMS)
   END_RUNG
   RUNG wire#powerrail
      Mul(in1 := "DB_Settings".InfeedToUpstreamEnableDelay, in2 := 1000.0, out => #"Time")
      { S7_Templates := "[SrcType := Real, DestType := DInt]" } Convert(in := #"Time", out => #InfeedToUpstreamEnableDelayMS)
   END_RUNG
   RUNG wire#powerrail
      Mul(in1 := "DB_Settings".OvercurrentSpinUpAllowance, in2 := 1000.0, out => #"Time")
      { S7_Templates := "[SrcType := Real, DestType := DInt]" } Convert(in := #"Time", out => #OvercurrentSpinUpAllowanceMS)
   END_RUNG
   RUNG wire#powerrail
      Mul(in1 := "DB_Settings".OvercurrentMediumDelay, in2 := 1000.0, out => #"Time")
      { S7_Templates := "[SrcType := Real, DestType := DInt]" } Convert(in := #"Time", out => #OvercurrentMediumDelayMS)
   END_RUNG
   RUNG wire#powerrail
      Mul(in1 := "DB_Settings".OvercurrentHighDelay, in2 := 1000.0, out => #"Time")
      { S7_Templates := "[SrcType := Real, DestType := DInt]" } Convert(in := #"Time", out => #OvercurrentHighDelayMS)
   END_RUNG
   RUNG wire#powerrail
      Mul(in1 := "DB_Settings".ReversalRetryPauseTime, in2 := 1000.0, out => #"Time")
      { S7_Templates := "[SrcType := Real, DestType := DInt]" } Convert(in := #"Time", out => #ReversalRetryPauseTimeMS)
   END_RUNG
   // the same network as SCL:
   #"Time" := "DB_Settings".ReversalWindowTime * 1000.0;
   #ReversalWindowTimeMS := REAL_TO_DINT(#"Time");
   #"Time" := "DB_Settings".PreStartSounderTime * 1000.0;
   #PreStartSounderTimeMS := REAL_TO_DINT(#"Time");
   #"Time" := "DB_Settings".DischargeConveyorTimeout * 1000.0;
   #DischargeConveyorTimeoutMS := REAL_TO_DINT(#"Time");
   #"Time" := "DB_Settings".ShredderReverseRunTime * 1000.0;
   #ShredderReverseRunTimeMS := REAL_TO_DINT(#"Time");
   #"Time" := "DB_Settings".InfeedRestartDelay * 1000.0;
   #InfeedRestartDelayMS := REAL_TO_DINT(#"Time");
   #"Time" := "DB_Settings".InfeedToUpstreamEnableDelay * 1000.0;
   #InfeedToUpstreamEnableDelayMS := REAL_TO_DINT(#"Time");
   #"Time" := "DB_Settings".OvercurrentSpinUpAllowance * 1000.0;
   #OvercurrentSpinUpAllowanceMS := REAL_TO_DINT(#"Time");
   #"Time" := "DB_Settings".OvercurrentMediumDelay * 1000.0;
   #OvercurrentMediumDelayMS := REAL_TO_DINT(#"Time");
   #"Time" := "DB_Settings".OvercurrentHighDelay * 1000.0;
   #OvercurrentHighDelayMS := REAL_TO_DINT(#"Time");
   #"Time" := "DB_Settings".ReversalRetryPauseTime * 1000.0;
   #ReversalRetryPauseTimeMS := REAL_TO_DINT(#"Time");
END_REGION

REGION Network 3: Reversal Re-Arm Window Timer
   // Retriggerable on-delay built from TON+edge. IN drops false the instant a NEW reversal is detected - Step transitioning into 60, tested against ReversalStepEdgeMem's own previous-scan value (correct read-before-write ordering: this network reads the memory bit before Network 4 updates it later the same scan, so no cross-network staleness) - which resets ET/Q to 0 that scan; the timer then re-arms and must run a full ReversalWindowTime with no further reversal before Q goes true.
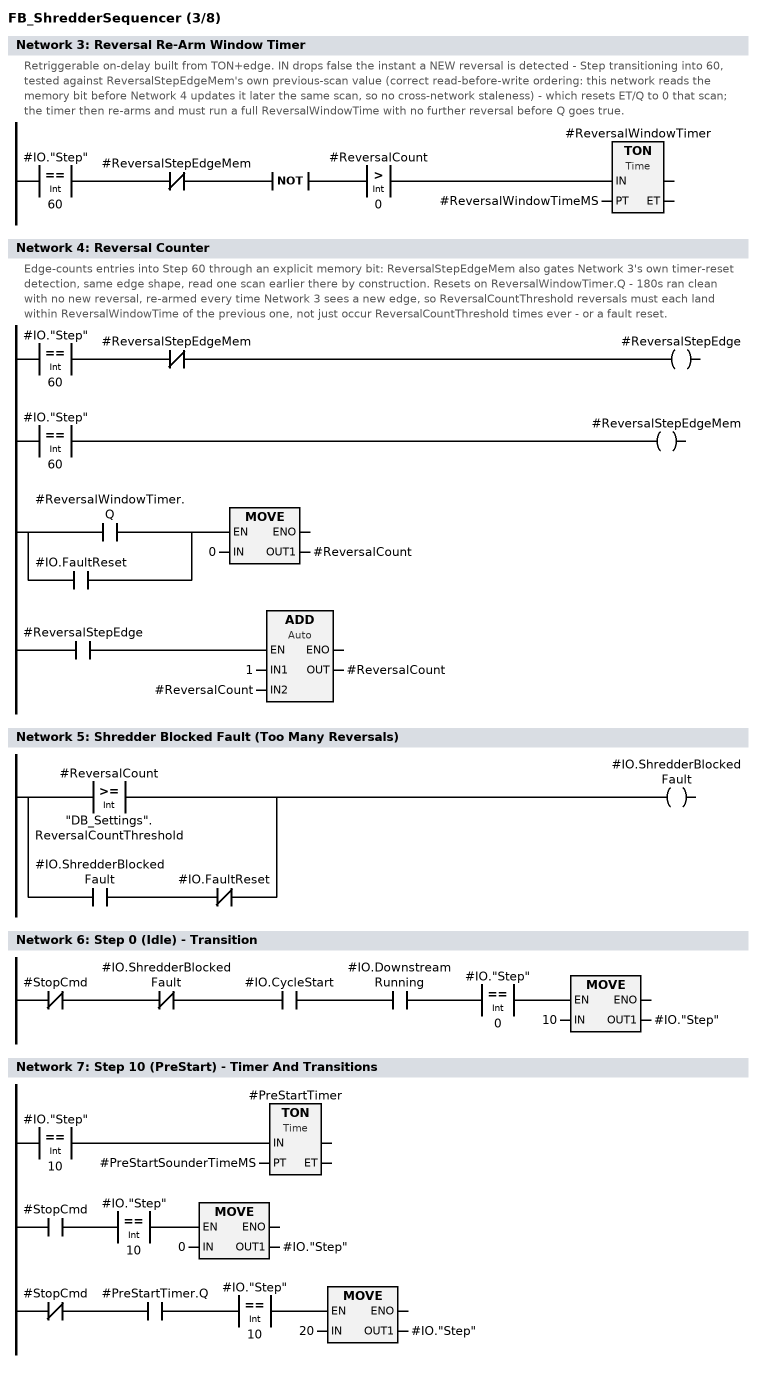
   RUNG wire#powerrail
      { S7_Templates := "SrcType := Int" } EQ_Contact(in1 := #IO."Step", in2 := 60)
      I_Contact( #ReversalStepEdgeMem )
      Not()
      { S7_Templates := "SrcType := Int" } GT_Contact(in1 := #ReversalCount, in2 := 0)
      { S7_Templates := "time_type := Time" } #ReversalWindowTimer.TON(pt := #ReversalWindowTimeMS, et =>)
   END_RUNG
   // the same network as SCL:
   #ReversalWindowTimer(IN := NOT ((#IO."Step" = 60) AND NOT #ReversalStepEdgeMem) AND (#ReversalCount > 0),   // TON
                        PT := #ReversalWindowTimeMS);
END_REGION

REGION Network 4: Reversal Counter
   // Edge-counts entries into Step 60 through an explicit memory bit: ReversalStepEdgeMem also gates Network 3's own timer-reset detection, same edge shape, read one scan earlier there by construction. Resets on ReversalWindowTimer.Q - 180s ran clean with no new reversal, re-armed every time Network 3 sees a new edge, so ReversalCountThreshold reversals must each land within ReversalWindowTime of the previous one, not just occur ReversalCountThreshold times ever - or a fault reset.
   RUNG wire#powerrail
      { S7_Templates := "SrcType := Int" } EQ_Contact(in1 := #IO."Step", in2 := 60)
      I_Contact( #ReversalStepEdgeMem )
      Coil( #ReversalStepEdge )
   END_RUNG
   RUNG wire#powerrail
      { S7_Templates := "SrcType := Int" } EQ_Contact(in1 := #IO."Step", in2 := 60)
      Coil( #ReversalStepEdgeMem )
   END_RUNG
   RUNG wire#powerrail
      Contact( #ReversalWindowTimer.Q )
      wire#w1
      Move(in := 0, out1 => #ReversalCount)
   END_RUNG
   RUNG wire#powerrail
      Contact( #IO.FaultReset )
   END_RUNG wire#w1
   RUNG wire#powerrail
      Contact( #ReversalStepEdge )
      Add(in1 := 1, in2 := #ReversalCount, out => #ReversalCount)
   END_RUNG
   // the same network as SCL:
   #ReversalStepEdge := (#IO."Step" = 60) AND NOT #ReversalStepEdgeMem;
   #ReversalStepEdgeMem := #IO."Step" = 60;
   IF #ReversalWindowTimer.Q OR #IO.FaultReset THEN #ReversalCount := 0; END_IF;
   IF #ReversalStepEdge THEN #ReversalCount := 1 + #ReversalCount; END_IF;
END_REGION

REGION Network 5: Shredder Blocked Fault (Too Many Reversals)
   RUNG wire#powerrail
      { S7_Templates := "SrcType := Int" } GE_Contact(in1 := #ReversalCount, in2 := "DB_Settings".ReversalCountThreshold)
      wire#w1
      Coil( #IO.ShredderBlockedFault )
   END_RUNG
   RUNG wire#powerrail
      Contact( #IO.ShredderBlockedFault )
      I_Contact( #IO.FaultReset )
   END_RUNG wire#w1
   // the same network as SCL:
   #IO.ShredderBlockedFault := (#ReversalCount >= "DB_Settings".ReversalCountThreshold) OR (#IO.ShredderBlockedFault AND NOT #IO.FaultReset);
END_REGION

REGION Network 6: Step 0 (Idle) - Transition
   RUNG wire#powerrail
      I_Contact( #StopCmd )
      I_Contact( #IO.ShredderBlockedFault )
      Contact( #IO.CycleStart )
      Contact( #IO.DownstreamRunning )
      { S7_Templates := "SrcType := Int" } EQ_Contact(in1 := #IO."Step", in2 := 0)
      Move(in := 10, out1 => #IO."Step")
   END_RUNG
   // the same network as SCL:
   IF NOT #StopCmd AND NOT #IO.ShredderBlockedFault AND #IO.CycleStart AND #IO.DownstreamRunning AND (#IO."Step" = 0) THEN
       #IO."Step" := 10;
   END_IF;
END_REGION

REGION Network 7: Step 10 (PreStart) - Timer And Transitions
   RUNG wire#powerrail
      { S7_Templates := "SrcType := Int" } EQ_Contact(in1 := #IO."Step", in2 := 10)
      { S7_Templates := "time_type := Time" } #PreStartTimer.TON(pt := #PreStartSounderTimeMS, et =>)
   END_RUNG
   RUNG wire#powerrail
      Contact( #StopCmd )
      { S7_Templates := "SrcType := Int" } EQ_Contact(in1 := #IO."Step", in2 := 10)
      Move(in := 0, out1 => #IO."Step")
   END_RUNG
   RUNG wire#powerrail
      I_Contact( #StopCmd )
      Contact( #PreStartTimer.Q )
      { S7_Templates := "SrcType := Int" } EQ_Contact(in1 := #IO."Step", in2 := 10)
      Move(in := 20, out1 => #IO."Step")
   END_RUNG
   // the same network as SCL:
   #PreStartTimer(IN := #IO."Step" = 10, PT := #PreStartSounderTimeMS);   // TON
   IF #StopCmd AND (#IO."Step" = 10) THEN #IO."Step" := 0; END_IF;
   IF NOT #StopCmd AND #PreStartTimer.Q AND (#IO."Step" = 10) THEN #IO."Step" := 20; END_IF;
END_REGION

REGION Network 8: Step 20 (DischargeStart) - Timer, Timeout Fault, And Transitions
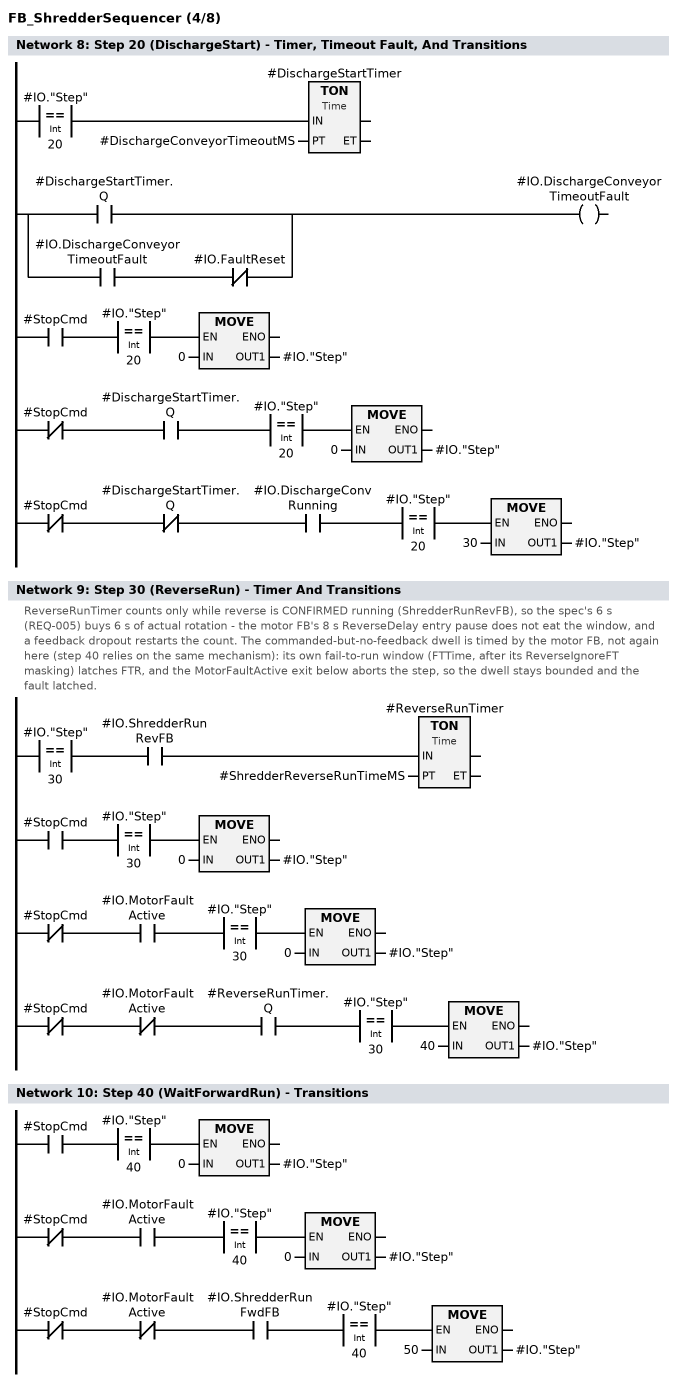
   RUNG wire#powerrail
      { S7_Templates := "SrcType := Int" } EQ_Contact(in1 := #IO."Step", in2 := 20)
      { S7_Templates := "time_type := Time" } #DischargeStartTimer.TON(pt := #DischargeConveyorTimeoutMS, et =>)
   END_RUNG
   RUNG wire#powerrail
      Contact( #DischargeStartTimer.Q )
      wire#w1
      Coil( #IO.DischargeConveyorTimeoutFault )
   END_RUNG
   RUNG wire#powerrail
      Contact( #IO.DischargeConveyorTimeoutFault )
      I_Contact( #IO.FaultReset )
   END_RUNG wire#w1
   RUNG wire#powerrail
      Contact( #StopCmd )
      { S7_Templates := "SrcType := Int" } EQ_Contact(in1 := #IO."Step", in2 := 20)
      Move(in := 0, out1 => #IO."Step")
   END_RUNG
   RUNG wire#powerrail
      I_Contact( #StopCmd )
      Contact( #DischargeStartTimer.Q )
      { S7_Templates := "SrcType := Int" } EQ_Contact(in1 := #IO."Step", in2 := 20)
      Move(in := 0, out1 => #IO."Step")
   END_RUNG
   RUNG wire#powerrail
      I_Contact( #StopCmd )
      I_Contact( #DischargeStartTimer.Q )
      Contact( #IO.DischargeConvRunning )
      { S7_Templates := "SrcType := Int" } EQ_Contact(in1 := #IO."Step", in2 := 20)
      Move(in := 30, out1 => #IO."Step")
   END_RUNG
   // the same network as SCL:
   #DischargeStartTimer(IN := #IO."Step" = 20, PT := #DischargeConveyorTimeoutMS);   // TON
   #IO.DischargeConveyorTimeoutFault := #DischargeStartTimer.Q OR (#IO.DischargeConveyorTimeoutFault AND NOT #IO.FaultReset);
   IF #StopCmd AND (#IO."Step" = 20) THEN #IO."Step" := 0; END_IF;
   IF NOT #StopCmd AND #DischargeStartTimer.Q AND (#IO."Step" = 20) THEN #IO."Step" := 0; END_IF;
   IF NOT #StopCmd AND NOT #DischargeStartTimer.Q AND #IO.DischargeConvRunning AND (#IO."Step" = 20) THEN
       #IO."Step" := 30;
   END_IF;
END_REGION

REGION Network 9: Step 30 (ReverseRun) - Timer And Transitions
   // ReverseRunTimer counts only while reverse is CONFIRMED running (ShredderRunRevFB), so the spec's 6 s (REQ-005) buys 6 s of actual rotation - the motor FB's 8 s ReverseDelay entry pause does not eat the window, and a feedback dropout restarts the count. The commanded-but-no-feedback dwell is timed by the motor FB, not again here (step 40 relies on the same mechanism): its own fail-to-run window (FTTime, after its ReverseIgnoreFT masking) latches FTR, and the MotorFaultActive exit below aborts the step, so the dwell stays bounded and the fault latched.
   RUNG wire#powerrail
      { S7_Templates := "SrcType := Int" } EQ_Contact(in1 := #IO."Step", in2 := 30)
      Contact( #IO.ShredderRunRevFB )
      { S7_Templates := "time_type := Time" } #ReverseRunTimer.TON(pt := #ShredderReverseRunTimeMS, et =>)
   END_RUNG
   RUNG wire#powerrail
      Contact( #StopCmd )
      { S7_Templates := "SrcType := Int" } EQ_Contact(in1 := #IO."Step", in2 := 30)
      Move(in := 0, out1 => #IO."Step")
   END_RUNG
   RUNG wire#powerrail
      I_Contact( #StopCmd )
      Contact( #IO.MotorFaultActive )
      { S7_Templates := "SrcType := Int" } EQ_Contact(in1 := #IO."Step", in2 := 30)
      Move(in := 0, out1 => #IO."Step")
   END_RUNG
   RUNG wire#powerrail
      I_Contact( #StopCmd )
      I_Contact( #IO.MotorFaultActive )
      Contact( #ReverseRunTimer.Q )
      { S7_Templates := "SrcType := Int" } EQ_Contact(in1 := #IO."Step", in2 := 30)
      Move(in := 40, out1 => #IO."Step")
   END_RUNG
   // the same network as SCL:
   #ReverseRunTimer(IN := (#IO."Step" = 30) AND #IO.ShredderRunRevFB, PT := #ShredderReverseRunTimeMS);   // TON
   IF #StopCmd AND (#IO."Step" = 30) THEN #IO."Step" := 0; END_IF;
   IF NOT #StopCmd AND #IO.MotorFaultActive AND (#IO."Step" = 30) THEN #IO."Step" := 0; END_IF;
   IF NOT #StopCmd AND NOT #IO.MotorFaultActive AND #ReverseRunTimer.Q AND (#IO."Step" = 30) THEN
       #IO."Step" := 40;
   END_IF;
END_REGION

REGION Network 10: Step 40 (WaitForwardRun) - Transitions
   RUNG wire#powerrail
      Contact( #StopCmd )
      { S7_Templates := "SrcType := Int" } EQ_Contact(in1 := #IO."Step", in2 := 40)
      Move(in := 0, out1 => #IO."Step")
   END_RUNG
   RUNG wire#powerrail
      I_Contact( #StopCmd )
      Contact( #IO.MotorFaultActive )
      { S7_Templates := "SrcType := Int" } EQ_Contact(in1 := #IO."Step", in2 := 40)
      Move(in := 0, out1 => #IO."Step")
   END_RUNG
   RUNG wire#powerrail
      I_Contact( #StopCmd )
      I_Contact( #IO.MotorFaultActive )
      Contact( #IO.ShredderRunFwdFB )
      { S7_Templates := "SrcType := Int" } EQ_Contact(in1 := #IO."Step", in2 := 40)
      Move(in := 50, out1 => #IO."Step")
   END_RUNG
   // the same network as SCL:
   IF #StopCmd AND (#IO."Step" = 40) THEN #IO."Step" := 0; END_IF;
   IF NOT #StopCmd AND #IO.MotorFaultActive AND (#IO."Step" = 40) THEN #IO."Step" := 0; END_IF;
   IF NOT #StopCmd AND NOT #IO.MotorFaultActive AND #IO.ShredderRunFwdFB AND (#IO."Step" = 40) THEN
       #IO."Step" := 50;
   END_IF;
END_REGION

REGION Network 11: Step 50 (Running) - Infeed Restart, Upstream Enable, And Outputs
   // UpstreamEnableTimer's own IN reads InfeedRunning one scan behind this network's own InfeedRunning update below (it's kind-ordered before the coil that writes it) - harmless for a multi-second delay. EnableUpstream lives here, next to its own timer, because it must only ever come from Step=50 dwell time, never from motor-running telemetry.
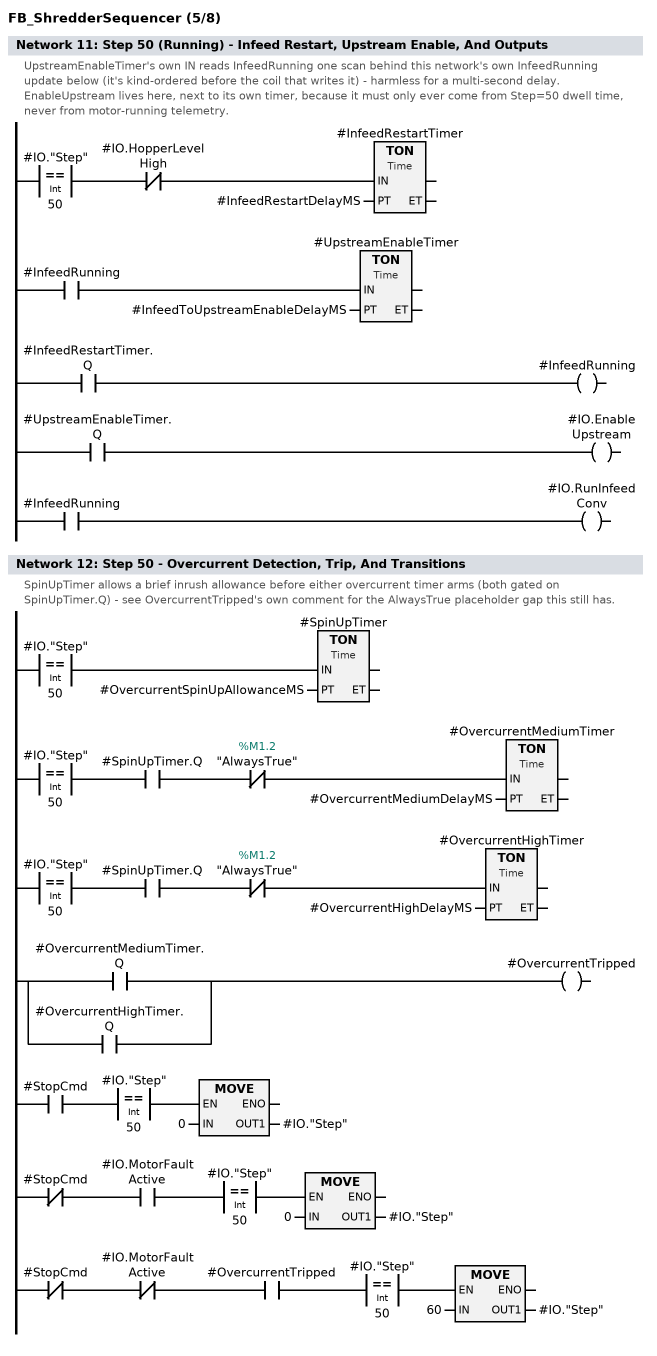
   RUNG wire#powerrail
      { S7_Templates := "SrcType := Int" } EQ_Contact(in1 := #IO."Step", in2 := 50)
      I_Contact( #IO.HopperLevelHigh )
      { S7_Templates := "time_type := Time" } #InfeedRestartTimer.TON(pt := #InfeedRestartDelayMS, et =>)
   END_RUNG
   RUNG wire#powerrail
      Contact( #InfeedRunning )
      { S7_Templates := "time_type := Time" } #UpstreamEnableTimer.TON(pt := #InfeedToUpstreamEnableDelayMS, et =>)
   END_RUNG
   RUNG wire#powerrail
      Contact( #InfeedRestartTimer.Q )
      Coil( #InfeedRunning )
   END_RUNG
   RUNG wire#powerrail
      Contact( #UpstreamEnableTimer.Q )
      Coil( #IO.EnableUpstream )
   END_RUNG
   RUNG wire#powerrail
      Contact( #InfeedRunning )
      Coil( #IO.RunInfeedConv )
   END_RUNG
   // the same network as SCL:
   #InfeedRestartTimer(IN := (#IO."Step" = 50) AND NOT #IO.HopperLevelHigh, PT := #InfeedRestartDelayMS);   // TON
   #UpstreamEnableTimer(IN := #InfeedRunning, PT := #InfeedToUpstreamEnableDelayMS);   // TON
   #InfeedRunning := #InfeedRestartTimer.Q;
   #IO.EnableUpstream := #UpstreamEnableTimer.Q;
   #IO.RunInfeedConv := #InfeedRunning;
END_REGION

REGION Network 12: Step 50 - Overcurrent Detection, Trip, And Transitions
   // SpinUpTimer allows a brief inrush allowance before either overcurrent timer arms (both gated on SpinUpTimer.Q) - see OvercurrentTripped's own comment for the AlwaysTrue placeholder gap this still has.
   RUNG wire#powerrail
      { S7_Templates := "SrcType := Int" } EQ_Contact(in1 := #IO."Step", in2 := 50)
      { S7_Templates := "time_type := Time" } #SpinUpTimer.TON(pt := #OvercurrentSpinUpAllowanceMS, et =>)
   END_RUNG
   RUNG wire#powerrail
      { S7_Templates := "SrcType := Int" } EQ_Contact(in1 := #IO."Step", in2 := 50)
      Contact( #SpinUpTimer.Q )
      I_Contact( "AlwaysTrue" )
      { S7_Templates := "time_type := Time" } #OvercurrentMediumTimer.TON(pt := #OvercurrentMediumDelayMS, et =>)
   END_RUNG
   RUNG wire#powerrail
      { S7_Templates := "SrcType := Int" } EQ_Contact(in1 := #IO."Step", in2 := 50)
      Contact( #SpinUpTimer.Q )
      I_Contact( "AlwaysTrue" )
      { S7_Templates := "time_type := Time" } #OvercurrentHighTimer.TON(pt := #OvercurrentHighDelayMS, et =>)
   END_RUNG
   RUNG wire#powerrail
      Contact( #OvercurrentMediumTimer.Q )
      wire#w1
      Coil( #OvercurrentTripped )
   END_RUNG
   RUNG wire#powerrail
      Contact( #OvercurrentHighTimer.Q )
   END_RUNG wire#w1
   RUNG wire#powerrail
      Contact( #StopCmd )
      { S7_Templates := "SrcType := Int" } EQ_Contact(in1 := #IO."Step", in2 := 50)
      Move(in := 0, out1 => #IO."Step")
   END_RUNG
   RUNG wire#powerrail
      I_Contact( #StopCmd )
      Contact( #IO.MotorFaultActive )
      { S7_Templates := "SrcType := Int" } EQ_Contact(in1 := #IO."Step", in2 := 50)
      Move(in := 0, out1 => #IO."Step")
   END_RUNG
   RUNG wire#powerrail
      I_Contact( #StopCmd )
      I_Contact( #IO.MotorFaultActive )
      Contact( #OvercurrentTripped )
      { S7_Templates := "SrcType := Int" } EQ_Contact(in1 := #IO."Step", in2 := 50)
      Move(in := 60, out1 => #IO."Step")
   END_RUNG
   // the same network as SCL:
   #SpinUpTimer(IN := #IO."Step" = 50, PT := #OvercurrentSpinUpAllowanceMS);   // TON
   #OvercurrentMediumTimer(IN := (#IO."Step" = 50) AND #SpinUpTimer.Q AND NOT "AlwaysTrue",   // TON
                           PT := #OvercurrentMediumDelayMS);
   #OvercurrentHighTimer(IN := (#IO."Step" = 50) AND #SpinUpTimer.Q AND NOT "AlwaysTrue",   // TON
                         PT := #OvercurrentHighDelayMS);
   #OvercurrentTripped := #OvercurrentMediumTimer.Q OR #OvercurrentHighTimer.Q;
   IF #StopCmd AND (#IO."Step" = 50) THEN #IO."Step" := 0; END_IF;
   IF NOT #StopCmd AND #IO.MotorFaultActive AND (#IO."Step" = 50) THEN #IO."Step" := 0; END_IF;
   IF NOT #StopCmd AND NOT #IO.MotorFaultActive AND #OvercurrentTripped AND (#IO."Step" = 50) THEN
       #IO."Step" := 60;
   END_IF;
END_REGION

REGION Network 13: Step 60 (OvercurrentAbort) - Timer And Transitions
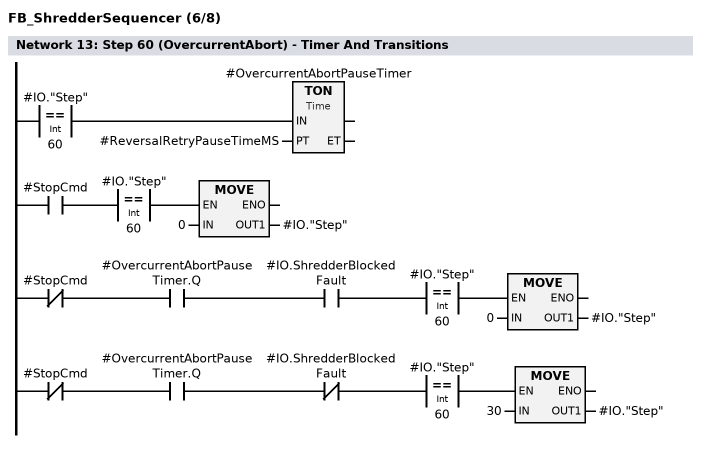
   RUNG wire#powerrail
      { S7_Templates := "SrcType := Int" } EQ_Contact(in1 := #IO."Step", in2 := 60)
      { S7_Templates := "time_type := Time" } #OvercurrentAbortPauseTimer.TON(pt := #ReversalRetryPauseTimeMS, et =>)
   END_RUNG
   RUNG wire#powerrail
      Contact( #StopCmd )
      { S7_Templates := "SrcType := Int" } EQ_Contact(in1 := #IO."Step", in2 := 60)
      Move(in := 0, out1 => #IO."Step")
   END_RUNG
   RUNG wire#powerrail
      I_Contact( #StopCmd )
      Contact( #OvercurrentAbortPauseTimer.Q )
      Contact( #IO.ShredderBlockedFault )
      { S7_Templates := "SrcType := Int" } EQ_Contact(in1 := #IO."Step", in2 := 60)
      Move(in := 0, out1 => #IO."Step")
   END_RUNG
   RUNG wire#powerrail
      I_Contact( #StopCmd )
      Contact( #OvercurrentAbortPauseTimer.Q )
      I_Contact( #IO.ShredderBlockedFault )
      { S7_Templates := "SrcType := Int" } EQ_Contact(in1 := #IO."Step", in2 := 60)
      Move(in := 30, out1 => #IO."Step")
   END_RUNG
   // the same network as SCL:
   #OvercurrentAbortPauseTimer(IN := #IO."Step" = 60, PT := #ReversalRetryPauseTimeMS);   // TON
   IF #StopCmd AND (#IO."Step" = 60) THEN #IO."Step" := 0; END_IF;
   IF NOT #StopCmd AND #OvercurrentAbortPauseTimer.Q AND #IO.ShredderBlockedFault AND (#IO."Step" = 60) THEN
       #IO."Step" := 0;
   END_IF;
   IF NOT #StopCmd AND #OvercurrentAbortPauseTimer.Q AND NOT #IO.ShredderBlockedFault AND (#IO."Step" = 60) THEN
       #IO."Step" := 30;
   END_IF;
END_REGION

REGION Network 14: Motor And Pusher Mode Commands
   // MotorStartArm asserts only through PreStart: one operator start press = one motor arming (FC_ControlMain hands it to the motor FB's self-clearing RecentStart - REQ-062). MotorReverseCmd is on for ReverseRun alone - Step 30 is the only step that runs the shredder backwards. MotorAutoStartCmd lists the steps that command the shredder motor to run - ReverseRun, WaitForwardRun and Running - and MotorPreStartDoneCmd lists the steps in which the pre-start warning already given still counts as in force - DischargeStart, ReverseRun, WaitForwardRun, Running and OvercurrentAbort; both list their steps individually, so a step added inside the cycle later has to decide for itself whether the motor is commanded during it and whether the warning still stands. OvercurrentAbort is one of the steps where it still stands: the abort pauses the cycle and resumes at ReverseRun without sounding the siren again (REQ-027), so the warning given at PreStart is still the warning in force through the pause, and the motor FB's pre-start memory stays latched across it. PusherParkCmd holds through the machine-start steps 20-40 as a range - any step inserted inside the start ramp still wants the pusher home - long enough for the pusher's warned repark to fire even when the discharge confirm is quick (REQ-045); from Running onward the pusher's own cycle-entry repark takes over. Pusher stop handling is two-tier (REQ-012/013): PusherModeForceOff (stop button/unhealthy/step-60, mirroring the step-60 overcurrent force) drives mode 0 - parks the pusher and blocks jog - while PusherCycleInhibitCmd mirrors the full StopCmd so downstream loss still stops cycle behavior without taking hand-jog away (REQ-040).
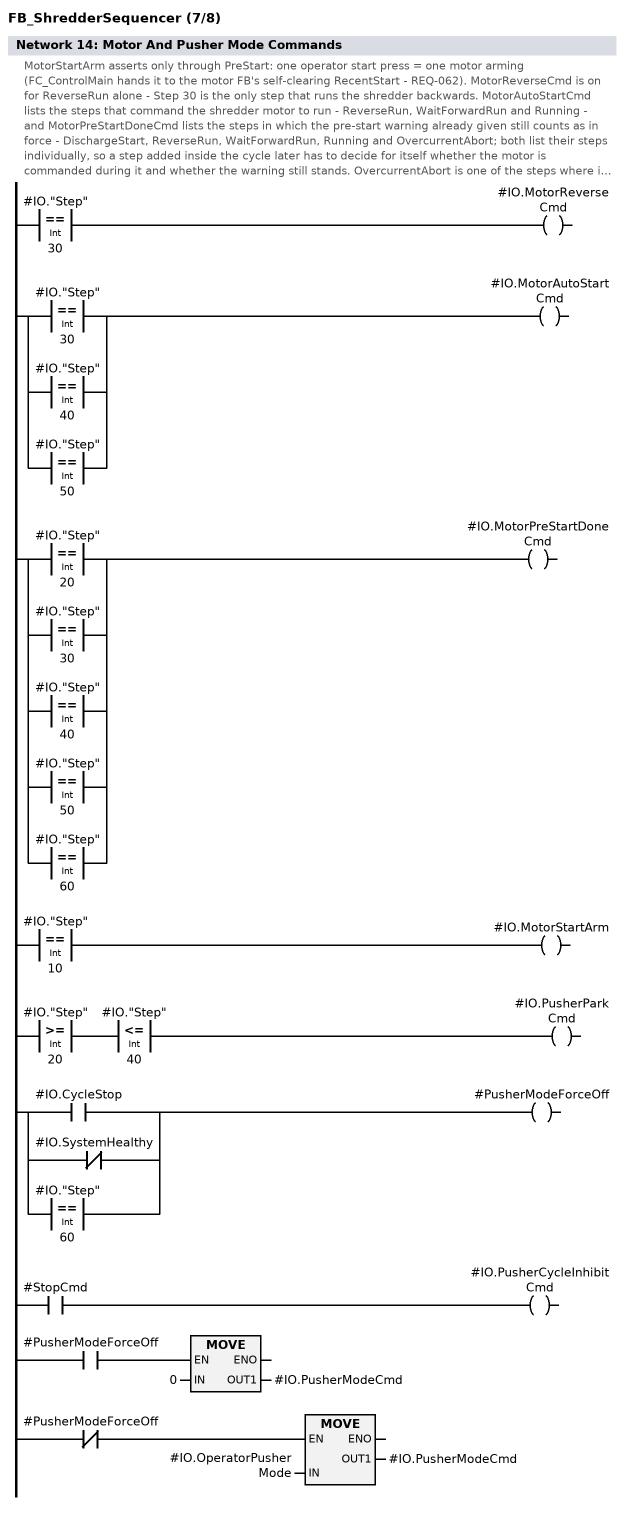
   RUNG wire#powerrail
      { S7_Templates := "SrcType := Int" } EQ_Contact(in1 := #IO."Step", in2 := 30)
      Coil( #IO.MotorReverseCmd )
   END_RUNG
   RUNG wire#powerrail
      { S7_Templates := "SrcType := Int" } EQ_Contact(in1 := #IO."Step", in2 := 30)
      wire#w1
      Coil( #IO.MotorAutoStartCmd )
   END_RUNG
   RUNG wire#powerrail
      { S7_Templates := "SrcType := Int" } EQ_Contact(in1 := #IO."Step", in2 := 40)
   END_RUNG wire#w1
   RUNG wire#powerrail
      { S7_Templates := "SrcType := Int" } EQ_Contact(in1 := #IO."Step", in2 := 50)
   END_RUNG wire#w1
   RUNG wire#powerrail
      { S7_Templates := "SrcType := Int" } EQ_Contact(in1 := #IO."Step", in2 := 20)
      wire#w2
      Coil( #IO.MotorPreStartDoneCmd )
   END_RUNG
   RUNG wire#powerrail
      { S7_Templates := "SrcType := Int" } EQ_Contact(in1 := #IO."Step", in2 := 30)
   END_RUNG wire#w2
   RUNG wire#powerrail
      { S7_Templates := "SrcType := Int" } EQ_Contact(in1 := #IO."Step", in2 := 40)
   END_RUNG wire#w2
   RUNG wire#powerrail
      { S7_Templates := "SrcType := Int" } EQ_Contact(in1 := #IO."Step", in2 := 50)
   END_RUNG wire#w2
   RUNG wire#powerrail
      { S7_Templates := "SrcType := Int" } EQ_Contact(in1 := #IO."Step", in2 := 60)
   END_RUNG wire#w2
   RUNG wire#powerrail
      { S7_Templates := "SrcType := Int" } EQ_Contact(in1 := #IO."Step", in2 := 10)
      Coil( #IO.MotorStartArm )
   END_RUNG
   RUNG wire#powerrail
      { S7_Templates := "SrcType := Int" } GE_Contact(in1 := #IO."Step", in2 := 20)
      { S7_Templates := "SrcType := Int" } LE_Contact(in1 := #IO."Step", in2 := 40)
      Coil( #IO.PusherParkCmd )
   END_RUNG
   RUNG wire#powerrail
      Contact( #IO.CycleStop )
      wire#w3
      Coil( #PusherModeForceOff )
   END_RUNG
   RUNG wire#powerrail
      I_Contact( #IO.SystemHealthy )
   END_RUNG wire#w3
   RUNG wire#powerrail
      { S7_Templates := "SrcType := Int" } EQ_Contact(in1 := #IO."Step", in2 := 60)
   END_RUNG wire#w3
   RUNG wire#powerrail
      Contact( #StopCmd )
      Coil( #IO.PusherCycleInhibitCmd )
   END_RUNG
   RUNG wire#powerrail
      Contact( #PusherModeForceOff )
      Move(in := 0, out1 => #IO.PusherModeCmd)
   END_RUNG
   RUNG wire#powerrail
      I_Contact( #PusherModeForceOff )
      Move(in := #IO.OperatorPusherMode, out1 => #IO.PusherModeCmd)
   END_RUNG
   // the same network as SCL:
   #IO.MotorReverseCmd := #IO."Step" = 30;
   #IO.MotorAutoStartCmd := (#IO."Step" = 30) OR (#IO."Step" = 40) OR (#IO."Step" = 50);
   #IO.MotorPreStartDoneCmd := (#IO."Step" = 20) OR (#IO."Step" = 30) OR (#IO."Step" = 40) OR (#IO."Step" = 50) OR (#IO."Step" = 60);
   #IO.MotorStartArm := #IO."Step" = 10;
   #IO.PusherParkCmd := (#IO."Step" >= 20) AND (#IO."Step" <= 40);
   #PusherModeForceOff := #IO.CycleStop OR NOT #IO.SystemHealthy OR (#IO."Step" = 60);
   #IO.PusherCycleInhibitCmd := #StopCmd;
   IF #PusherModeForceOff THEN #IO.PusherModeCmd := 0; END_IF;
   IF NOT #PusherModeForceOff THEN #IO.PusherModeCmd := #IO.OperatorPusherMode; END_IF;
END_REGION

REGION Network 15: Output Commands
   // Cycle output commands: the discharge conveyor runs during DischargeStart, ReverseRun, WaitForwardRun, Running and OvercurrentAbort, each step on its own branch, so a step added inside the cycle later has to decide for itself whether the conveyor runs during it; the pre-start siren sounds during PreStart or whenever the pusher asks for its own jog warning; and InCycle reports any step other than Idle.
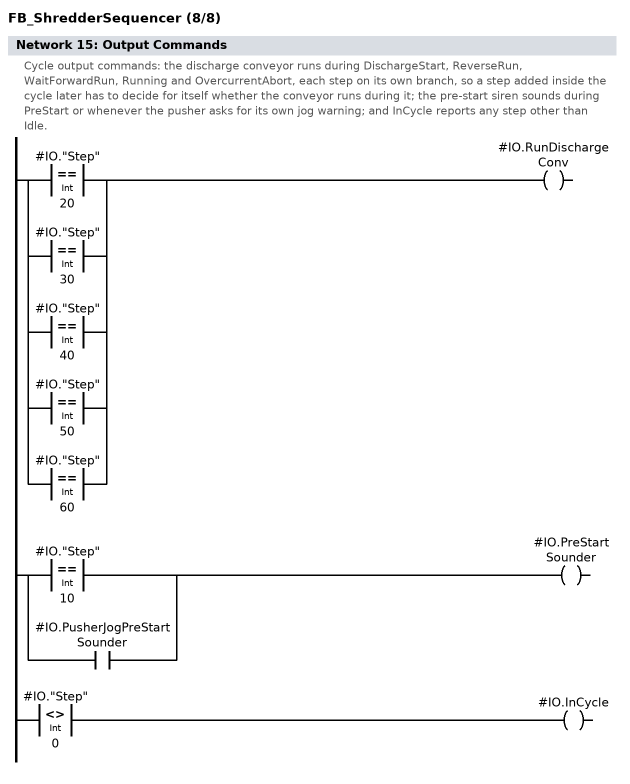
   RUNG wire#powerrail
      { S7_Templates := "SrcType := Int" } EQ_Contact(in1 := #IO."Step", in2 := 20)
      wire#w1
      Coil( #IO.RunDischargeConv )
   END_RUNG
   RUNG wire#powerrail
      { S7_Templates := "SrcType := Int" } EQ_Contact(in1 := #IO."Step", in2 := 30)
   END_RUNG wire#w1
   RUNG wire#powerrail
      { S7_Templates := "SrcType := Int" } EQ_Contact(in1 := #IO."Step", in2 := 40)
   END_RUNG wire#w1
   RUNG wire#powerrail
      { S7_Templates := "SrcType := Int" } EQ_Contact(in1 := #IO."Step", in2 := 50)
   END_RUNG wire#w1
   RUNG wire#powerrail
      { S7_Templates := "SrcType := Int" } EQ_Contact(in1 := #IO."Step", in2 := 60)
   END_RUNG wire#w1
   RUNG wire#powerrail
      { S7_Templates := "SrcType := Int" } EQ_Contact(in1 := #IO."Step", in2 := 10)
      wire#w2
      Coil( #IO.PreStartSounder )
   END_RUNG
   RUNG wire#powerrail
      Contact( #IO.PusherJogPreStartSounder )
   END_RUNG wire#w2
   RUNG wire#powerrail
      { S7_Templates := "SrcType := Int" } NE_Contact(in1 := #IO."Step", in2 := 0)
      Coil( #IO.InCycle )
   END_RUNG
   // the same network as SCL:
   #IO.RunDischargeConv := (#IO."Step" = 20) OR (#IO."Step" = 30) OR (#IO."Step" = 40) OR (#IO."Step" = 50) OR (#IO."Step" = 60);
   #IO.PreStartSounder := (#IO."Step" = 10) OR #IO.PusherJogPreStartSounder;
   #IO.InCycle := #IO."Step" <> 0;
END_REGION
END_FUNCTION_BLOCK

FUNCTION_BLOCK "FB_PusherControl"   // FB3, LAD
TITLE = Pusher Control
{ S7_Optimized_Access := 'TRUE' }
VERSION : 0.1
// Pusher ram sequencing (C-118-C-125). Step legend (C-120): 0=Idle (no motion; home is the HomeLimit switch, not implied by the step - after a jog release the ram may legitimately rest off home, REQ-039) - 10=DriveToEndTravel (forward stroke in progress) - 20=Hold (paused at full travel, brief settle before retracting) - 30=Retract (returning to home; also the recovery/abort target from any bad state). Mode legend: 0=Off (finish a retract already in progress, then park; no new cycle starts) - 1=Auto (hopper-high-level starts a cycle) - 2=Manual (operator button/jog starts a cycle). Motion policy (owner rulings 2026-07-16): an idle off-home ram reparks ONLY on the plant pre-start ParkCmd or on a live cycle request - never on jog release or bare mode changes - and every motion start from rest (repark, cycle launch, jog) is preceded by the JogWarningTime sounder warning (NEW-4: no unwarned pusher motion). CycleInhibit (any live plant stop reason) blocks cycle launches and aborts an in-flight cycle to park, but deliberately leaves hand-jog available - only the mode-0 force (stop button/unhealthy) blocks jogging (owner amendment 2026-07-16, REQ-040). Fitted=FALSE (REQ-042/043/044) kills every demand, the pack output, both supervision timers, and every fault latch at the source, so a disabled pusher does nothing and raises nothing.
// stored: AutoNumber true, IsIECCheckEnabled false, IsRetainMemResEnabled false, MemoryReserve 100, SetENOAutomatically false, UDAEnableTagReadback false
   VAR RETAIN
      IO { S7_SetPoint := 'True'} : "UDT_PusherIO";   // Caller-visible interface (C-115) - FC_ControlMain writes Mode/HopperHighLevel/limits/tunables in, reads Extend/Retract/RunPowerPack/fault bits out. See the block header for the Step/Mode value legend.
   END_VAR
   VAR
      CycleRequest : Bool;   // Named once, read everywhere (C-601): the live cycle trigger - Auto on hopper high or Manual on the HMI button - gated by Enable (Fitted AND not Off) and NOT Blocked. Read by the warning armer, the launch and repark transitions, and the trip-count reset. Blocked is written later in the scan, so this reads it one scan behind - immaterial: Blocked can only latch mid-stroke (Step 10) where no Step 0 request can act, and a reset-clear merely delays a relaunch by one scan.
      JogDemand : Bool;   // A live jog request: either jog button held, idle, Manual mode, pusher fitted. Arms the pre-motion warning, suppresses the repark (jogging is never fought by an auto-retract), and - per direction, warning done - drives the demands. Reads Step from before this scan's transitions; the demand rungs re-check Step fresh.
      ReparkRequest : Bool;   // A repark to home is wanted: the sequencer's pre-start ParkCmd (REQ-045) or a live CycleRequest, while idle off home and not jogging. One of the only two motion sources out of Step 0 (owner ruling 2026-07-16); fires the 0-to-30 transition once the pre-motion warning has sounded.
      LaunchRequest : Bool;   // A cycle launch is possible: live CycleRequest, idle, ram at home. Fires the 0-to-10 transition once the pre-motion warning has sounded; the same fired condition resets PressureTripCount (per-cycle jam counting, REQ-048).
      CycleAbort : Bool;   // Named once (C-601): abort an in-flight cycle to Retract - Off commanded mid-cycle, or the plant acquired a stop reason (CycleInhibit). Read by the Step 10 and Step 20 exits; the Step 30 retract completes regardless, so an aborted cycle always ends parked. Jog is untouched by this bit (owner amendment 2026-07-16).
      EndTravelTimeoutMS : DInt;
      ParkedTimeoutMS : DInt;
      EndTravelHoldTimeMS : DInt;
      PumpRunOnTimeMS : DInt;
      JogWarningTimeMS : DInt;
      PressureTripConfirmTimeMS : DInt;
      PressureClearResumeDelayMS : DInt;
      PressureConfirmTimer { S7_SetPoint := 'True'} : TON_TIME;
      PressureClearTimer { S7_SetPoint := 'True'} : TON_TIME;
      PressureHold : Bool;   // Latched jam hold, not a fault (C-123) - see the Pressure Detection network. Freezes ExtendDemand while set; clears itself once pressure has genuinely stayed clear for PressureClearResumeDelay.
      PressureConfirmEdge : Bool;
      PressureConfirmEdgeMem : Bool;
      PressureTripCount : Int;   // Confirmed jams this cycle - reset each cycle start, not time-windowed. Compared against IO.PressureTripCountThreshold to raise Blocked.
      EndTravelTimer { S7_SetPoint := 'True'} : TON_TIME;
      HoldTimer { S7_SetPoint := 'True'} : TON_TIME;
      ParkedTimer { S7_SetPoint := 'True'} : TON_TIME;
      JogPreStartTimer { S7_SetPoint := 'True'} : TON_TIME;
      ExtendDemand : Bool;
      RetractDemand : Bool;
      PumpDemand : Bool;   // ExtendDemand OR RetractDemand - the pump's own immediate (non-run-on) demand signal.
      PumpEverDemanded : Bool;   // Cold-start guard for the pump run-on off-delay below - see that network's own comment.
      PumpRunOnTimer { S7_SetPoint := 'True'} : TON_TIME;
   END_VAR
   VAR_TEMP
      "Time" : Real;
   END_VAR
BEGIN

REGION Network 1: Enable And Motion Requests
   // The compound conditions every later network shares, each written once (C-601). Requests read Step as it settled last scan (the transitions run later) - safe, because Step only ever leaves 0 through this scan's own request-gated transitions; steps returning to 0 just re-arm the requests one scan late. CycleInhibit kills cycle requests (no launch into a stopped plant) and, via CycleAbort, retracts an in-flight cycle - while JogDemand deliberately ignores it: hand-jog stays available with the plant stopped by downstream absence (owner amendment 2026-07-16, REQ-040).
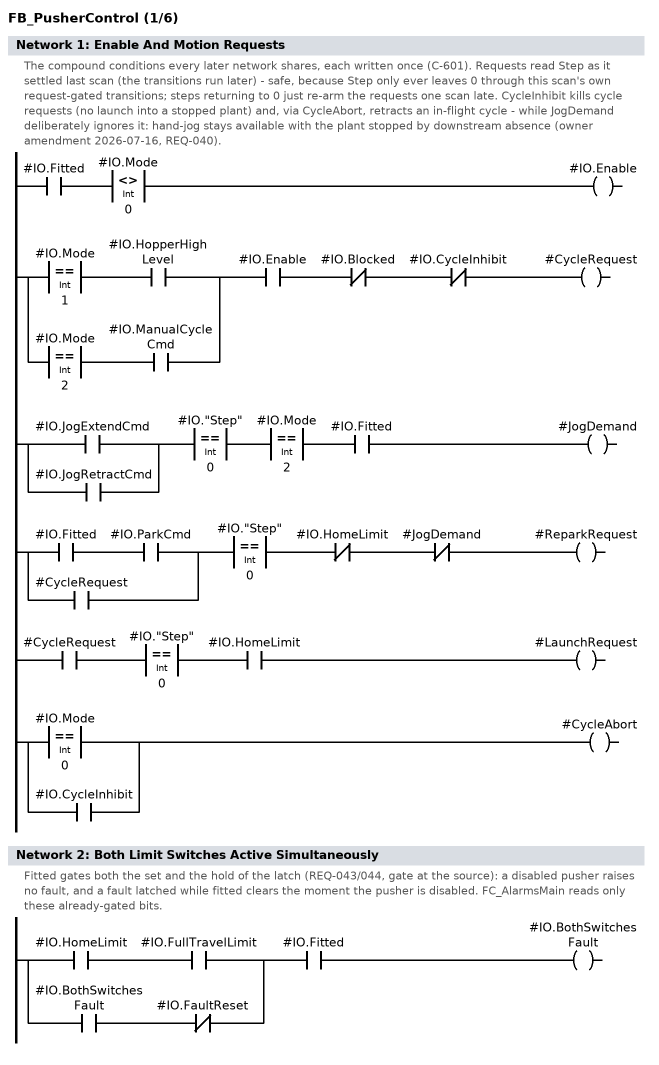
   RUNG wire#powerrail
      Contact( #IO.Fitted )
      { S7_Templates := "SrcType := Int" } NE_Contact(in1 := #IO.Mode, in2 := 0)
      Coil( #IO.Enable )
   END_RUNG
   RUNG wire#powerrail
      { S7_Templates := "SrcType := Int" } EQ_Contact(in1 := #IO.Mode, in2 := 1)
      Contact( #IO.HopperHighLevel )
      wire#w1
      Contact( #IO.Enable )
      I_Contact( #IO.Blocked )
      I_Contact( #IO.CycleInhibit )
      Coil( #CycleRequest )
   END_RUNG
   RUNG wire#powerrail
      { S7_Templates := "SrcType := Int" } EQ_Contact(in1 := #IO.Mode, in2 := 2)
      Contact( #IO.ManualCycleCmd )
   END_RUNG wire#w1
   RUNG wire#powerrail
      Contact( #IO.JogExtendCmd )
      wire#w2
      { S7_Templates := "SrcType := Int" } EQ_Contact(in1 := #IO."Step", in2 := 0)
      { S7_Templates := "SrcType := Int" } EQ_Contact(in1 := #IO.Mode, in2 := 2)
      Contact( #IO.Fitted )
      Coil( #JogDemand )
   END_RUNG
   RUNG wire#powerrail
      Contact( #IO.JogRetractCmd )
   END_RUNG wire#w2
   RUNG wire#powerrail
      Contact( #IO.Fitted )
      Contact( #IO.ParkCmd )
      wire#w3
      { S7_Templates := "SrcType := Int" } EQ_Contact(in1 := #IO."Step", in2 := 0)
      I_Contact( #IO.HomeLimit )
      I_Contact( #JogDemand )
      Coil( #ReparkRequest )
   END_RUNG
   RUNG wire#powerrail
      Contact( #CycleRequest )
   END_RUNG wire#w3
   RUNG wire#powerrail
      Contact( #CycleRequest )
      { S7_Templates := "SrcType := Int" } EQ_Contact(in1 := #IO."Step", in2 := 0)
      Contact( #IO.HomeLimit )
      Coil( #LaunchRequest )
   END_RUNG
   RUNG wire#powerrail
      { S7_Templates := "SrcType := Int" } EQ_Contact(in1 := #IO.Mode, in2 := 0)
      wire#w4
      Coil( #CycleAbort )
   END_RUNG
   RUNG wire#powerrail
      Contact( #IO.CycleInhibit )
   END_RUNG wire#w4
   // the same network as SCL:
   #IO.Enable := #IO.Fitted AND (#IO.Mode <> 0);
   #CycleRequest := (((#IO.Mode = 1) AND #IO.HopperHighLevel) OR ((#IO.Mode = 2) AND #IO.ManualCycleCmd)) AND #IO.Enable AND NOT #IO.Blocked AND NOT #IO.CycleInhibit;
   #JogDemand := (#IO.JogExtendCmd OR #IO.JogRetractCmd) AND (#IO."Step" = 0) AND (#IO.Mode = 2) AND #IO.Fitted;
   #ReparkRequest := ((#IO.Fitted AND #IO.ParkCmd) OR #CycleRequest) AND (#IO."Step" = 0) AND NOT #IO.HomeLimit AND NOT #JogDemand;
   #LaunchRequest := #CycleRequest AND (#IO."Step" = 0) AND #IO.HomeLimit;
   #CycleAbort := (#IO.Mode = 0) OR #IO.CycleInhibit;
END_REGION

REGION Network 2: Both Limit Switches Active Simultaneously
   // Fitted gates both the set and the hold of the latch (REQ-043/044, gate at the source): a disabled pusher raises no fault, and a fault latched while fitted clears the moment the pusher is disabled. FC_AlarmsMain reads only these already-gated bits.
   RUNG wire#powerrail
      Contact( #IO.HomeLimit )
      Contact( #IO.FullTravelLimit )
      wire#w1
      Contact( #IO.Fitted )
      Coil( #IO.BothSwitchesFault )
   END_RUNG
   RUNG wire#powerrail
      Contact( #IO.BothSwitchesFault )
      I_Contact( #IO.FaultReset )
   END_RUNG wire#w1
   // the same network as SCL:
   #IO.BothSwitchesFault := ((#IO.HomeLimit AND #IO.FullTravelLimit) OR (#IO.BothSwitchesFault AND NOT #IO.FaultReset)) AND #IO.Fitted;
END_REGION

REGION Network 3: HMI Time Conversions
   // HMI/DB_Settings times are Real seconds for operator legibility; every TON below needs its PT in DInt ms - one MUL+CONVERT pair per timer, matching the MotorDOL FTTime/EnableUPSTime idiom. Kept as one block up front rather than repeated at each timer, so the x1000 idiom is visibly consistent and only ever done once.
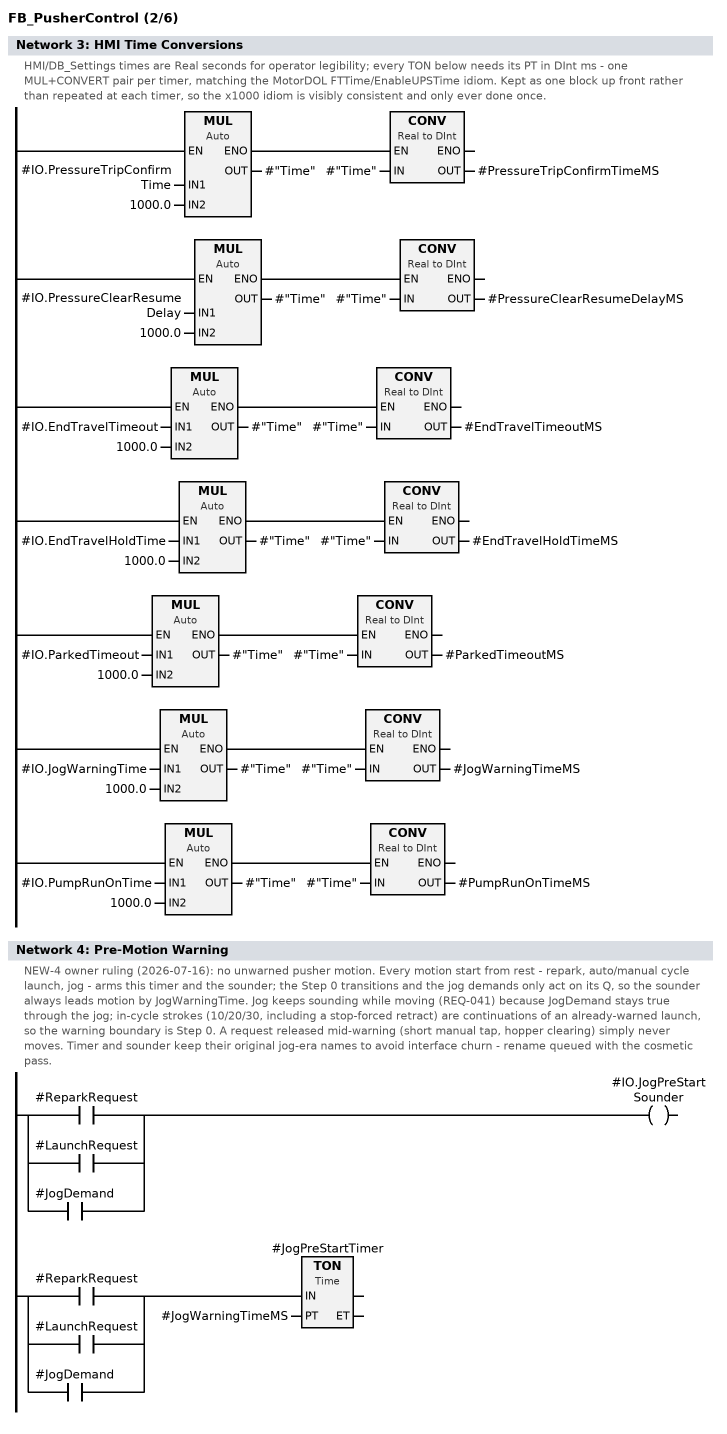
   RUNG wire#powerrail
      Mul(in1 := #IO.PressureTripConfirmTime, in2 := 1000.0, out => #"Time")
      { S7_Templates := "[SrcType := Real, DestType := DInt]" } Convert(in := #"Time", out => #PressureTripConfirmTimeMS)
   END_RUNG
   RUNG wire#powerrail
      Mul(in1 := #IO.PressureClearResumeDelay, in2 := 1000.0, out => #"Time")
      { S7_Templates := "[SrcType := Real, DestType := DInt]" } Convert(in := #"Time", out => #PressureClearResumeDelayMS)
   END_RUNG
   RUNG wire#powerrail
      Mul(in1 := #IO.EndTravelTimeout, in2 := 1000.0, out => #"Time")
      { S7_Templates := "[SrcType := Real, DestType := DInt]" } Convert(in := #"Time", out => #EndTravelTimeoutMS)
   END_RUNG
   RUNG wire#powerrail
      Mul(in1 := #IO.EndTravelHoldTime, in2 := 1000.0, out => #"Time")
      { S7_Templates := "[SrcType := Real, DestType := DInt]" } Convert(in := #"Time", out => #EndTravelHoldTimeMS)
   END_RUNG
   RUNG wire#powerrail
      Mul(in1 := #IO.ParkedTimeout, in2 := 1000.0, out => #"Time")
      { S7_Templates := "[SrcType := Real, DestType := DInt]" } Convert(in := #"Time", out => #ParkedTimeoutMS)
   END_RUNG
   RUNG wire#powerrail
      Mul(in1 := #IO.JogWarningTime, in2 := 1000.0, out => #"Time")
      { S7_Templates := "[SrcType := Real, DestType := DInt]" } Convert(in := #"Time", out => #JogWarningTimeMS)
   END_RUNG
   RUNG wire#powerrail
      Mul(in1 := #IO.PumpRunOnTime, in2 := 1000.0, out => #"Time")
      { S7_Templates := "[SrcType := Real, DestType := DInt]" } Convert(in := #"Time", out => #PumpRunOnTimeMS)
   END_RUNG
   // the same network as SCL:
   #"Time" := #IO.PressureTripConfirmTime * 1000.0;
   #PressureTripConfirmTimeMS := REAL_TO_DINT(#"Time");
   #"Time" := #IO.PressureClearResumeDelay * 1000.0;
   #PressureClearResumeDelayMS := REAL_TO_DINT(#"Time");
   #"Time" := #IO.EndTravelTimeout * 1000.0;
   #EndTravelTimeoutMS := REAL_TO_DINT(#"Time");
   #"Time" := #IO.EndTravelHoldTime * 1000.0;
   #EndTravelHoldTimeMS := REAL_TO_DINT(#"Time");
   #"Time" := #IO.ParkedTimeout * 1000.0;
   #ParkedTimeoutMS := REAL_TO_DINT(#"Time");
   #"Time" := #IO.JogWarningTime * 1000.0;
   #JogWarningTimeMS := REAL_TO_DINT(#"Time");
   #"Time" := #IO.PumpRunOnTime * 1000.0;
   #PumpRunOnTimeMS := REAL_TO_DINT(#"Time");
END_REGION

REGION Network 4: Pre-Motion Warning
   // NEW-4 owner ruling (2026-07-16): no unwarned pusher motion. Every motion start from rest - repark, auto/manual cycle launch, jog - arms this timer and the sounder; the Step 0 transitions and the jog demands only act on its Q, so the sounder always leads motion by JogWarningTime. Jog keeps sounding while moving (REQ-041) because JogDemand stays true through the jog; in-cycle strokes (10/20/30, including a stop-forced retract) are continuations of an already-warned launch, so the warning boundary is Step 0. A request released mid-warning (short manual tap, hopper clearing) simply never moves. Timer and sounder keep their original jog-era names to avoid interface churn - rename queued with the cosmetic pass.
   RUNG wire#powerrail
      Contact( #ReparkRequest )
      wire#w1
      Coil( #IO.JogPreStartSounder )
   END_RUNG
   RUNG wire#powerrail
      Contact( #LaunchRequest )
   END_RUNG wire#w1
   RUNG wire#powerrail
      Contact( #JogDemand )
   END_RUNG wire#w1
   RUNG wire#powerrail
      Contact( #ReparkRequest )
      wire#w2
      { S7_Templates := "time_type := Time" } #JogPreStartTimer.TON(pt := #JogWarningTimeMS, et =>)
   END_RUNG
   RUNG wire#powerrail
      Contact( #LaunchRequest )
   END_RUNG wire#w2
   RUNG wire#powerrail
      Contact( #JogDemand )
   END_RUNG wire#w2
   // the same network as SCL:
   #IO.JogPreStartSounder := #ReparkRequest OR #LaunchRequest OR #JogDemand;
   #JogPreStartTimer(IN := #ReparkRequest OR #LaunchRequest OR #JogDemand, PT := #JogWarningTimeMS);   // TON
END_REGION

REGION Network 5: Pressure Trip Detection, Hold, And Counting
   // One function, one network: a trip must be debounced (PressureConfirmTimer) before it counts - momentary pressure spikes aren't a real jam. Hold latches through a confirmed trip and only releases once pressure has genuinely cleared for PressureClearResumeDelay, so a bouncing switch can't re-trigger the count on every scan. Count resets each cycle start (the same LaunchRequest-and-warning-done condition that fires the 0-to-10 launch), not on a rolling time window.
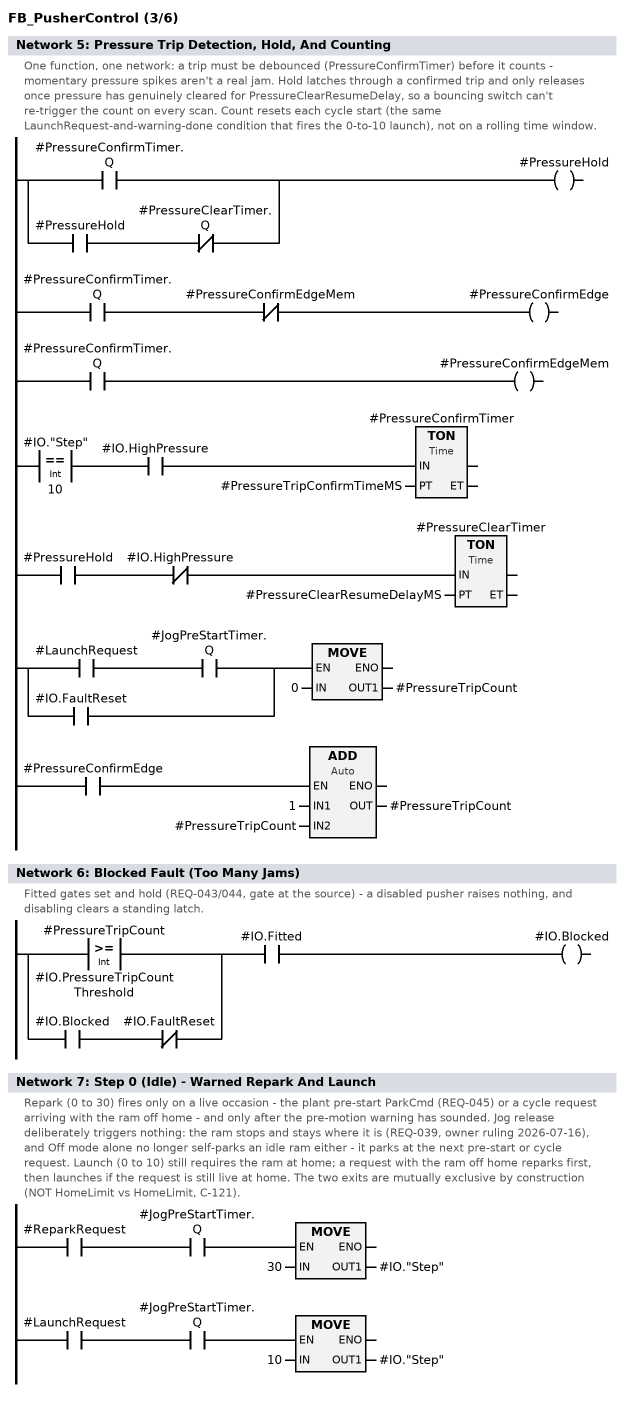
   RUNG wire#powerrail
      Contact( #PressureConfirmTimer.Q )
      wire#w1
      Coil( #PressureHold )
   END_RUNG
   RUNG wire#powerrail
      Contact( #PressureHold )
      I_Contact( #PressureClearTimer.Q )
   END_RUNG wire#w1
   RUNG wire#powerrail
      Contact( #PressureConfirmTimer.Q )
      I_Contact( #PressureConfirmEdgeMem )
      Coil( #PressureConfirmEdge )
   END_RUNG
   RUNG wire#powerrail
      Contact( #PressureConfirmTimer.Q )
      Coil( #PressureConfirmEdgeMem )
   END_RUNG
   RUNG wire#powerrail
      { S7_Templates := "SrcType := Int" } EQ_Contact(in1 := #IO."Step", in2 := 10)
      Contact( #IO.HighPressure )
      { S7_Templates := "time_type := Time" } #PressureConfirmTimer.TON(pt := #PressureTripConfirmTimeMS, et =>)
   END_RUNG
   RUNG wire#powerrail
      Contact( #PressureHold )
      I_Contact( #IO.HighPressure )
      { S7_Templates := "time_type := Time" } #PressureClearTimer.TON(pt := #PressureClearResumeDelayMS, et =>)
   END_RUNG
   RUNG wire#powerrail
      Contact( #LaunchRequest )
      Contact( #JogPreStartTimer.Q )
      wire#w2
      Move(in := 0, out1 => #PressureTripCount)
   END_RUNG
   RUNG wire#powerrail
      Contact( #IO.FaultReset )
   END_RUNG wire#w2
   RUNG wire#powerrail
      Contact( #PressureConfirmEdge )
      Add(in1 := 1, in2 := #PressureTripCount, out => #PressureTripCount)
   END_RUNG
   // the same network as SCL:
   #PressureHold := #PressureConfirmTimer.Q OR (#PressureHold AND NOT #PressureClearTimer.Q);
   #PressureConfirmEdge := #PressureConfirmTimer.Q AND NOT #PressureConfirmEdgeMem;
   #PressureConfirmEdgeMem := #PressureConfirmTimer.Q;
   #PressureConfirmTimer(IN := (#IO."Step" = 10) AND #IO.HighPressure, PT := #PressureTripConfirmTimeMS);   // TON
   #PressureClearTimer(IN := #PressureHold AND NOT #IO.HighPressure, PT := #PressureClearResumeDelayMS);   // TON
   IF (#LaunchRequest AND #JogPreStartTimer.Q) OR #IO.FaultReset THEN #PressureTripCount := 0; END_IF;
   IF #PressureConfirmEdge THEN #PressureTripCount := 1 + #PressureTripCount; END_IF;
END_REGION

REGION Network 6: Blocked Fault (Too Many Jams)
   // Fitted gates set and hold (REQ-043/044, gate at the source) - a disabled pusher raises nothing, and disabling clears a standing latch.
   RUNG wire#powerrail
      { S7_Templates := "SrcType := Int" } GE_Contact(in1 := #PressureTripCount, in2 := #IO.PressureTripCountThreshold)
      wire#w1
      Contact( #IO.Fitted )
      Coil( #IO.Blocked )
   END_RUNG
   RUNG wire#powerrail
      Contact( #IO.Blocked )
      I_Contact( #IO.FaultReset )
   END_RUNG wire#w1
   // the same network as SCL:
   #IO.Blocked := ((#PressureTripCount >= #IO.PressureTripCountThreshold) OR (#IO.Blocked AND NOT #IO.FaultReset)) AND #IO.Fitted;
END_REGION

